LIN {X 0,Y 410.175,Z 395.355,A -85,B 0,C 180,E1 -10523.613,E2 -10523.613} C_VEL
LIN {X 0,Y 410.092,Z 398.974,A -85,B 0,C 180,E1 -10525.084,E2 -10525.084} C_VEL
LIN {X 0,Y 409.955,Z 400.845,A -85,B 0,C 180,E1 -10526.067,E2 -10526.067} C_VEL
LIN {X 0,Y 409.994,Z 402.256,A -85,B 0,C 180,E1 -10527.052,E2 -10527.052} C_VEL
LIN {X 0,Y 409.99,Z 403.255,A -85,B 0,C 180,E1 -10528.035,E2 -10528.035} C_VEL
LIN {X 0,Y 409.957,Z 404.069,A -85,B 0,C 180,E1 -10529.999,E2 -10529.999} C_VEL
LIN {X 0,Y 409.949,Z 403.838,A -85,B 0,C 180,E1 -10530.982,E2 -10530.982} C_VEL
LIN {X 0,Y 409.99,Z 403.212,A -85,B 0,C 180,E1 -10531.964,E2 -10531.964} C_VEL
LIN {X 0,Y 410.009,Z 402.191,A -85,B 0,C 180,E1 -10532.947,E2 -10532.947} C_VEL
LIN {X 0,Y 409.956,Z 400.758,A -85,B 0,C 180,E1 -10533.931,E2 -10533.931} C_VEL
LIN {X 0,Y 410.11,Z 397.769,A -85,B 0,C 180,E1 -10535.408,E2 -10535.408} C_VEL
LIN {X 0,Y 410.201,Z 393.722,A -85,B 0,C 180,E1 -10536.888,E2 -10536.888} C_VEL
LIN {X 0,Y 410.553,Z 387.517,A -85,B 0,C 180,E1 -10538.614,E2 -10538.614} C_VEL
LIN {X 0,Y 410.987,Z 380.75,A -85,B 0,C 180,E1 -10540.094,E2 -10540.094} C_VEL
LIN {X 0,Y 411.568,Z 372.368,A -85,B 0,C 180,E1 -10541.574,E2 -10541.574} C_VEL
LIN {X 0,Y 412.213,Z 363.785,A -85,B 0,C 180,E1 -10542.805,E2 -10542.805} C_VEL
LIN {X 0,Y 412.957,Z 353.054,A -85,B 0,C 180,E1 -10544.051,E2 -10544.051} C_VEL
LIN {X 0,Y 413.774,Z 341.349,A -85,B 0,C 180,E1 -10545.137,E2 -10545.137} C_VEL
LIN {X 0,Y 414.645,Z 329.481,A -85,B 0,C 180,E1 -10545.986,E2 -10545.986} C_VEL
LIN {X 0,Y 414.751,Z 323.251,A -85,B 0,C 180,E1 -10546.359,E2 -10546.359} C_VEL
LIN {X 0,Y 412.959,Z 310.23,A -85,B 0,C 180,E1 -10547.058,E2 -10547.058} C_VEL
LIN {X 0,Y 410.902,Z 297.191,A -85,B 0,C 180,E1 -10547.565,E2 -10547.565} C_VEL
LIN {X 0,Y 410.692,Z 295.43,A -85,B 0,C 180,E1 -10547.629,E2 -10547.629} C_VEL
LIN {X 0,Y 410.997,Z 287.996,A -85,B 0,C 180,E1 -10550.52,E2 -10550.52} C_VEL
LIN {X 0,Y 411.365,Z 280.065,A -85,B 0,C 180,E1 -10553.67,E2 -10553.67} C_VEL
LIN {X 0,Y 411.926,Z 270.899,A -85,B 0,C 180,E1 -10557.429,E2 -10557.429} C_VEL
LIN {X 0,Y 412.494,Z 263.176,A -85,B 0,C 180,E1 -10560.739,E2 -10560.739} C_VEL
LIN {X 0,Y 413.163,Z 255.633,A -85,B 0,C 180,E1 -10564.147,E2 -10564.147} C_VEL
LIN {X 0,Y 413.517,Z 251.98,A -85,B 0,C 180,E1 -10565.897,E2 -10565.897} C_VEL
LIN {X 0,Y 413.199,Z 248.334,A -85,B 0,C 180,E1 -10567.756,E2 -10567.756} C_VEL
LIN {X 0,Y 412.06,Z 241.871,A -85,B 0,C 180,E1 -10571.369,E2 -10571.369} C_VEL
LIN {X 0,Y 411.195,Z 237.269,A -85,B 0,C 180,E1 -10574.262,E2 -10574.262} C_VEL
LIN {X 0,Y 411.193,Z 237.266,A -85,B 0,C 180,E1 -10577.301,E2 -10577.301} C_VEL
LIN {X 0,Y 411.232,Z 237.264,A -85,B 0,C 180,E1 -10580.776,E2 -10580.776} C_VEL
LIN {X 0,Y 411.2,Z 237.268,A -85,B 0,C 180,E1 -10584.47,E2 -10584.47} C_VEL
LIN {X 0,Y 411.207,Z 237.264,A -85,B 0,C 180,E1 -10586.872,E2 -10586.872} C_VEL
LIN {X 0,Y 411.233,Z 237.26,A -85,B 0,C 180,E1 -10590.643,E2 -10590.643} C_VEL
LIN {X 0,Y 411.238,Z 237.261,A -85,B 0,C 180,E1 -10593.618,E2 -10593.618} C_VEL
LIN {X 0,Y 411.202,Z 237.265,A -85,B 0,C 180,E1 -10596.851,E2 -10596.851} C_VEL
LIN {X 0,Y 411.214,Z 237.261,A -85,B 0,C 180,E1 -10600.049,E2 -10600.049} C_VEL
LIN {X 0,Y 411.261,Z 237.258,A -85,B 0,C 180,E1 -10603.13,E2 -10603.13} C_VEL
LIN {X 0,Y 411.303,Z 237.251,A -85,B 0,C 180,E1 -10606.894,E2 -10606.894} C_VEL
LIN {X 0,Y 411.29,Z 237.255,A -85,B 0,C 180,E1 -10610.16,E2 -10610.16} C_VEL
LIN {X 0,Y 411.458,Z 237.233,A -85,B 0,C 180,E1 -10613.131,E2 -10613.131} C_VEL
LIN {X 0,Y 411.309,Z 237.252,A -85,B 0,C 180,E1 -10615.097,E2 -10615.097} C_VEL
LIN {X 0,Y 411.51,Z 237.226,A -85,B 0,C 180,E1 -10618.041,E2 -10618.041} C_VEL
LIN {X 0,Y 411.64,Z 237.211,A -85,B 0,C 180,E1 -10619.998,E2 -10619.998} C_VEL
LIN {X 0,Y 411.461,Z 237.233,A -85,B 0,C 180,E1 -10622.936,E2 -10622.936} C_VEL
LIN {X 0,Y 411.455,Z 237.236,A -85,B 0,C 180,E1 -10626.865,E2 -10626.865} C_VEL
LIN {X 0,Y 411.345,Z 237.249,A -85,B 0,C 180,E1 -10628.844,E2 -10628.844} C_VEL
LIN {X 0,Y 411.165,Z 237.277,A -85,B 0,C 180,E1 -10631.834,E2 -10631.834} C_VEL
LIN {X 0,Y 411.052,Z 237.291,A -85,B 0,C 180,E1 -10632.955,E2 -10632.955} C_VEL
LIN {X 0,Y 410.907,Z 240.592,A -85,B 0,C 180,E1 -10636.707,E2 -10636.707} C_VEL
LIN {X 0,Y 410.742,Z 243.677,A -85,B 0,C 180,E1 -10640.009,E2 -10640.009} C_VEL
LIN {X 0,Y 410.621,Z 246.692,A -85,B 0,C 180,E1 -10643.18,E2 -10643.18} C_VEL
LIN {X 0,Y 410.51,Z 249.844,A -85,B 0,C 180,E1 -10646.429,E2 -10646.429} C_VEL
LIN {X 0,Y 410.442,Z 252.871,A -85,B 0,C 180,E1 -10649.486,E2 -10649.486} C_VEL
LIN {X 0,Y 414.108,Z 266.327,A -85,B 0,C 180,E1 -10650.146,E2 -10650.146} C_VEL
LIN {X 0,Y 415.728,Z 274.254,A -85,B 0,C 180,E1 -10650.613,E2 -10650.613} C_VEL
LIN {X 0,Y 415.069,Z 286.599,A -85,B 0,C 180,E1 -10651.374,E2 -10651.374} C_VEL
LIN {X 0,Y 414.368,Z 298.089,A -85,B 0,C 180,E1 -10652.296,E2 -10652.296} C_VEL
LIN {X 0,Y 413.578,Z 309.114,A -85,B 0,C 180,E1 -10653.422,E2 -10653.422} C_VEL
LIN {X 0,Y 412.865,Z 318.531,A -85,B 0,C 180,E1 -10654.617,E2 -10654.617} C_VEL
LIN {X 0,Y 412.164,Z 327.573,A -85,B 0,C 180,E1 -10656.032,E2 -10656.032} C_VEL
LIN {X 0,Y 411.605,Z 334.198,A -85,B 0,C 180,E1 -10657.308,E2 -10657.308} C_VEL
LIN {X 0,Y 411.016,Z 341.072,A -85,B 0,C 180,E1 -10658.966,E2 -10658.966} C_VEL
LIN {X 0,Y 410.659,Z 346.195,A -85,B 0,C 180,E1 -10660.564,E2 -10660.564} C_VEL
LIN {X 0,Y 410.323,Z 350.805,A -85,B 0,C 180,E1 -10662.567,E2 -10662.567} C_VEL
LIN {X 0,Y 410.109,Z 352.955,A -85,B 0,C 180,E1 -10663.967,E2 -10663.967} C_VEL
LIN {X 0,Y 410.013,Z 354.243,A -85,B 0,C 180,E1 -10665.351,E2 -10665.351} C_VEL
LIN {X 0,Y 409.943,Z 354.715,A -85,B 0,C 180,E1 -10666.706,E2 -10666.706} C_VEL
LIN {X 0,Y 409.959,Z 354.458,A -85,B 0,C 180,E1 -10668.043,E2 -10668.043} C_VEL
LIN {X 0,Y 410.031,Z 353.501,A -85,B 0,C 180,E1 -10669.359,E2 -10669.359} C_VEL
LIN {X 0,Y 410.218,Z 350.71,A -85,B 0,C 180,E1 -10671.294,E2 -10671.294} C_VEL
LIN {X 0,Y 410.512,Z 346.397,A -85,B 0,C 180,E1 -10673.188,E2 -10673.188} C_VEL
LIN {X 0,Y 410.875,Z 341.126,A -85,B 0,C 180,E1 -10674.839,E2 -10674.839} C_VEL
LIN {X 0,Y 411.274,Z 335.33,A -85,B 0,C 180,E1 -10676.265,E2 -10676.265} C_VEL
LIN {X 0,Y 411.887,Z 327.667,A -85,B 0,C 180,E1 -10677.778,E2 -10677.778} C_VEL
LIN {X 0,Y 412.441,Z 320.075,A -85,B 0,C 180,E1 -10679,E2 -10679} C_VEL
LIN {X 0,Y 413.135,Z 310.353,A -85,B 0,C 180,E1 -10680.281,E2 -10680.281} C_VEL
LIN {X 0,Y 413.83,Z 300.496,A -85,B 0,C 180,E1 -10681.331,E2 -10681.331} C_VEL
LIN {X 0,Y 414.563,Z 288.332,A -85,B 0,C 180,E1 -10682.369,E2 -10682.369} C_VEL
LIN {X 0,Y 415.22,Z 276.391,A -85,B 0,C 180,E1 -10683.147,E2 -10683.147} C_VEL
LIN {X 0,Y 415.328,Z 272.584,A -85,B 0,C 180,E1 -10683.358,E2 -10683.358} C_VEL
LIN {X 0,Y 412.637,Z 260.388,A -85,B 0,C 180,E1 -10684.022,E2 -10684.022} C_VEL
LIN {X 0,Y 410.354,Z 251.228,A -85,B 0,C 180,E1 -10684.446,E2 -10684.446} C_VEL
LIN {X 0,Y 410.359,Z 247.606,A -85,B 0,C 180,E1 -10687.866,E2 -10687.866} C_VEL
LIN {X 0,Y 410.438,Z 244.343,A -85,B 0,C 180,E1 -10691.014,E2 -10691.014} C_VEL
LIN {X 0,Y 410.537,Z 241.175,A -85,B 0,C 180,E1 -10694.104,E2 -10694.104} C_VEL
LIN {X 0,Y 410.648,Z 237.964,A -85,B 0,C 180,E1 -10697.285,E2 -10697.285} C_VEL
LIN {X 0,Y 410.713,Z 237.33,A -85,B 0,C 180,E1 -10698.151,E2 -10698.151} C_VEL
LIN {X 0,Y 411.121,Z 237.277,A -85,B 0,C 180,E1 -10701.15,E2 -10701.15} C_VEL
LIN {X 0,Y 411.4,Z 237.241,A -85,B 0,C 180,E1 -10703.133,E2 -10703.133} C_VEL
LIN {X 0,Y 411.299,Z 237.254,A -85,B 0,C 180,E1 -10705.099,E2 -10705.099} C_VEL
LIN {X 0,Y 411.498,Z 237.227,A -85,B 0,C 180,E1 -10708.043,E2 -10708.043} C_VEL
LIN {X 0,Y 411.626,Z 237.21,A -85,B 0,C 180,E1 -10710.006,E2 -10710.006} C_VEL
LIN {X 0,Y 411.452,Z 237.234,A -85,B 0,C 180,E1 -10712.938,E2 -10712.938} C_VEL
LIN {X 0,Y 411.244,Z 237.257,A -85,B 0,C 180,E1 -10714.283,E2 -10714.283} C_VEL
LIN {X 0,Y 410.636,Z 237.337,A -85,B 0,C 180,E1 -10715.101,E2 -10715.101} C_VEL
LIN {X 0,Y 407.876,Z 237.677,A -85,B 0,C 180,E1 -10716.434,E2 -10716.434} C_VEL
LIN {X 0,Y 405.488,Z 237.977,A -85,B 0,C 180,E1 -10717.51,E2 -10717.51} C_VEL
LIN {X 0,Y 404.421,Z 238.107,A -85,B 0,C 180,E1 -10718.34,E2 -10718.34} C_VEL
LIN {X 0,Y 404.314,Z 238.121,A -85,B 0,C 180,E1 -10718.622,E2 -10718.622} C_VEL
LIN {X 0,Y 404.255,Z 238.127,A -85,B 0,C 180,E1 -10722.042,E2 -10722.042} C_VEL
LIN {X 0,Y 404.192,Z 238.139,A -85,B 0,C 180,E1 -10725.119,E2 -10725.119} C_VEL
LIN {X 0,Y 404.199,Z 238.135,A -85,B 0,C 180,E1 -10728.239,E2 -10728.239} C_VEL
LIN {X 0,Y 404.18,Z 238.139,A -85,B 0,C 180,E1 -10731.418,E2 -10731.418} C_VEL
LIN {X 0,Y 404.165,Z 238.143,A -85,B 0,C 180,E1 -10734.667,E2 -10734.667} C_VEL
LIN {X 0,Y 404.182,Z 238.137,A -85,B 0,C 180,E1 -10738.001,E2 -10738.001} C_VEL
LIN {X 0,Y 404.127,Z 238.144,A -85,B 0,C 180,E1 -10741.56,E2 -10741.56} C_VEL
LIN {X 0,Y 404.174,Z 238.141,A -85,B 0,C 180,E1 -10745.018,E2 -10745.018} C_VEL
LIN {X 0,Y 404.153,Z 238.145,A -85,B 0,C 180,E1 -10748.758,E2 -10748.758} C_VEL
LIN {X 0,Y 404.181,Z 238.137,A -85,B 0,C 180,E1 -10751.613,E2 -10751.613} C_VEL
LIN {X 0,Y 404.19,Z 238.14,A -85,B 0,C 180,E1 -10754.532,E2 -10754.532} C_VEL
LIN {X 0,Y 404.202,Z 238.135,A -85,B 0,C 180,E1 -10757.307,E2 -10757.307} C_VEL
LIN {X 0,Y 404.161,Z 238.142,A -85,B 0,C 180,E1 -10759.957,E2 -10759.957} C_VEL
LIN {X 0,Y 404.134,Z 238.143,A -85,B 0,C 180,E1 -10763.126,E2 -10763.126} C_VEL
LIN {X 0,Y 404.139,Z 238.146,A -85,B 0,C 180,E1 -10766.19,E2 -10766.19} C_VEL
LIN {X 0,Y 404.15,Z 238.143,A -85,B 0,C 180,E1 -10769.718,E2 -10769.718} C_VEL
LIN {X 0,Y 404.191,Z 238.135,A -85,B 0,C 180,E1 -10773.125,E2 -10773.125} C_VEL
LIN {X 0,Y 404.174,Z 238.138,A -85,B 0,C 180,E1 -10775.336,E2 -10775.336} C_VEL
LIN {X 0,Y 404.136,Z 238.144,A -85,B 0,C 180,E1 -10778.583,E2 -10778.583} C_VEL
LIN {X 0,Y 404.209,Z 238.136,A -85,B 0,C 180,E1 -10781.764,E2 -10781.764} C_VEL
LIN {X 0,Y 404.205,Z 238.134,A -85,B 0,C 180,E1 -10784.884,E2 -10784.884} C_VEL
LIN {X 0,Y 404.256,Z 238.132,A -85,B 0,C 180,E1 -10787.96,E2 -10787.96} C_VEL
LIN {X 0,Y 404.266,Z 238.126,A -85,B 0,C 180,E1 -10791,E2 -10791} C_VEL
LIN {X 0,Y 404.418,Z 238.112,A -85,B 0,C 180,E1 -10794.017,E2 -10794.017} C_VEL
LIN {X 0,Y 404.482,Z 238.103,A -85,B 0,C 180,E1 -10798.01,E2 -10798.01} C_VEL
LIN {X 0,Y 404.612,Z 238.087,A -85,B 0,C 180,E1 -10800.002,E2 -10800.002} C_VEL
LIN {X 0,Y 404.417,Z 238.108,A -85,B 0,C 180,E1 -10802.99,E2 -10802.99} C_VEL
LIN {X 0,Y 404.373,Z 238.114,A -85,B 0,C 180,E1 -10806.989,E2 -10806.989} C_VEL
LIN {X 0,Y 404.261,Z 238.13,A -85,B 0,C 180,E1 -10810.013,E2 -10810.013} C_VEL
LIN {X 0,Y 404.272,Z 238.128,A -85,B 0,C 180,E1 -10813.213,E2 -10813.213} C_VEL
LIN {X 0,Y 404.221,Z 238.134,A -85,B 0,C 180,E1 -10817.008,E2 -10817.008} C_VEL
LIN {X 0,Y 404.17,Z 238.139,A -85,B 0,C 180,E1 -10820.353,E2 -10820.353} C_VEL
LIN {X 0,Y 404.171,Z 238.143,A -85,B 0,C 180,E1 -10823.576,E2 -10823.576} C_VEL
LIN {X 0,Y 404.187,Z 238.139,A -85,B 0,C 180,E1 -10825.768,E2 -10825.768} C_VEL
LIN {X 0,Y 404.201,Z 238.135,A -85,B 0,C 180,E1 -10828.001,E2 -10828.001} C_VEL
LIN {X 0,Y 404.145,Z 238.145,A -85,B 0,C 180,E1 -10831.559,E2 -10831.559} C_VEL
LIN {X 0,Y 404.19,Z 238.14,A -85,B 0,C 180,E1 -10835.017,E2 -10835.017} C_VEL
LIN {X 0,Y 404.158,Z 238.143,A -85,B 0,C 180,E1 -10838.758,E2 -10838.758} C_VEL
LIN {X 0,Y 404.129,Z 238.145,A -85,B 0,C 180,E1 -10841.6,E2 -10841.6} C_VEL
LIN {X 0,Y 404.152,Z 238.141,A -85,B 0,C 180,E1 -10844.522,E2 -10844.522} C_VEL
LIN {X 0,Y 404.163,Z 238.245,A -85,B 0,C 180,E1 -10846.106,E2 -10846.106} C_VEL
LIN {X 0,Y 405.086,Z 243.048,A -85,B 0,C 180,E1 -10848.755,E2 -10848.755} C_VEL
LIN {X 0,Y 406.008,Z 248.19,A -85,B 0,C 180,E1 -10851.452,E2 -10851.452} C_VEL
LIN {X 0,Y 406.492,Z 252.053,A -85,B 0,C 180,E1 -10853.381,E2 -10853.381} C_VEL
LIN {X 0,Y 406.251,Z 257.069,A -85,B 0,C 180,E1 -10855.73,E2 -10855.73} C_VEL
LIN {X 0,Y 405.685,Z 263.641,A -85,B 0,C 180,E1 -10858.686,E2 -10858.686} C_VEL
LIN {X 0,Y 405.074,Z 271.812,A -85,B 0,C 180,E1 -10862.234,E2 -10862.234} C_VEL
LIN {X 0,Y 404.464,Z 280.525,A -85,B 0,C 180,E1 -10865.899,E2 -10865.899} C_VEL
LIN {X 0,Y 404.05,Z 288.356,A -85,B 0,C 180,E1 -10869.11,E2 -10869.11} C_VEL
LIN {X 0,Y 403.652,Z 295.818,A -85,B 0,C 180,E1 -10872.096,E2 -10872.096} C_VEL
LIN {X 0,Y 405.932,Z 309.766,A -85,B 0,C 180,E1 -10872.631,E2 -10872.631} C_VEL
LIN {X 0,Y 407.729,Z 322.632,A -85,B 0,C 180,E1 -10873.322,E2 -10873.322} C_VEL
LIN {X 0,Y 407.99,Z 325.826,A -85,B 0,C 180,E1 -10873.516,E2 -10873.516} C_VEL
LIN {X 0,Y 407.131,Z 338.126,A -85,B 0,C 180,E1 -10874.352,E2 -10874.352} C_VEL
LIN {X 0,Y 406.279,Z 349.865,A -85,B 0,C 180,E1 -10875.383,E2 -10875.383} C_VEL
LIN {X 0,Y 405.613,Z 359.75,A -85,B 0,C 180,E1 -10876.472,E2 -10876.472} C_VEL
LIN {X 0,Y 404.877,Z 368.986,A -85,B 0,C 180,E1 -10877.722,E2 -10877.722} C_VEL
LIN {X 0,Y 404.108,Z 377.981,A -85,B 0,C 180,E1 -10879.224,E2 -10879.224} C_VEL
LIN {X 0,Y 403.616,Z 385.238,A -85,B 0,C 180,E1 -10880.731,E2 -10880.731} C_VEL
LIN {X 0,Y 403.305,Z 390.139,A -85,B 0,C 180,E1 -10881.986,E2 -10881.986} C_VEL
LIN {X 0,Y 403.068,Z 395.38,A -85,B 0,C 180,E1 -10883.658,E2 -10883.658} C_VEL
LIN {X 0,Y 403.004,Z 398.551,A -85,B 0,C 180,E1 -10884.997,E2 -10884.997} C_VEL
LIN {X 0,Y 402.877,Z 400.424,A -85,B 0,C 180,E1 -10885.998,E2 -10885.998} C_VEL
LIN {X 0,Y 402.897,Z 401.835,A -85,B 0,C 180,E1 -10887,E2 -10887} C_VEL
LIN {X 0,Y 402.922,Z 402.836,A -85,B 0,C 180,E1 -10888,E2 -10888} C_VEL
LIN {X 0,Y 402.881,Z 403.647,A -85,B 0,C 180,E1 -10889.999,E2 -10889.999} C_VEL
LIN {X 0,Y 402.876,Z 403.417,A -85,B 0,C 180,E1 -10890.999,E2 -10890.999} C_VEL
LIN {X 0,Y 402.923,Z 402.79,A -85,B 0,C 180,E1 -10891.999,E2 -10891.999} C_VEL
LIN {X 0,Y 402.91,Z 401.764,A -85,B 0,C 180,E1 -10892.999,E2 -10892.999} C_VEL
LIN {X 0,Y 402.879,Z 400.331,A -85,B 0,C 180,E1 -10894.001,E2 -10894.001} C_VEL
LIN {X 0,Y 403.008,Z 397.336,A -85,B 0,C 180,E1 -10895.503,E2 -10895.503} C_VEL
LIN {X 0,Y 403.12,Z 393.285,A -85,B 0,C 180,E1 -10897.009,E2 -10897.009} C_VEL
LIN {X 0,Y 403.519,Z 387.077,A -85,B 0,C 180,E1 -10898.765,E2 -10898.765} C_VEL
LIN {X 0,Y 403.962,Z 380.309,A -85,B 0,C 180,E1 -10900.272,E2 -10900.272} C_VEL
LIN {X 0,Y 404.577,Z 371.931,A -85,B 0,C 180,E1 -10901.777,E2 -10901.777} C_VEL
LIN {X 0,Y 405.236,Z 363.356,A -85,B 0,C 180,E1 -10903.029,E2 -10903.029} C_VEL
LIN {X 0,Y 405.984,Z 353.509,A -85,B 0,C 180,E1 -10904.203,E2 -10904.203} C_VEL
LIN {X 0,Y 406.781,Z 342.376,A -85,B 0,C 180,E1 -10905.276,E2 -10905.276} C_VEL
LIN {X 0,Y 407.662,Z 331.108,A -85,B 0,C 180,E1 -10906.133,E2 -10906.133} C_VEL
LIN {X 0,Y 407.911,Z 324.517,A -85,B 0,C 180,E1 -10906.549,E2 -10906.549} C_VEL
LIN {X 0,Y 406.181,Z 311.546,A -85,B 0,C 180,E1 -10907.284,E2 -10907.284} C_VEL
LIN {X 0,Y 404.207,Z 298.69,A -85,B 0,C 180,E1 -10907.827,E2 -10907.827} C_VEL
LIN {X 0,Y 403.633,Z 294.95,A -85,B 0,C 180,E1 -10907.969,E2 -10907.969} C_VEL
LIN {X 0,Y 403.947,Z 287.608,A -85,B 0,C 180,E1 -10910.895,E2 -10910.895} C_VEL
LIN {X 0,Y 404.356,Z 279.728,A -85,B 0,C 180,E1 -10914.107,E2 -10914.107} C_VEL
LIN {X 0,Y 404.94,Z 271.136,A -85,B 0,C 180,E1 -10917.73,E2 -10917.73} C_VEL
LIN {X 0,Y 405.485,Z 264.205,A -85,B 0,C 180,E1 -10920.75,E2 -10920.75} C_VEL
LIN {X 0,Y 406.177,Z 256.624,A -85,B 0,C 180,E1 -10924.264,E2 -10924.264} C_VEL
LIN {X 0,Y 406.511,Z 251.844,A -85,B 0,C 180,E1 -10926.616,E2 -10926.616} C_VEL
LIN {X 0,Y 405.905,Z 247.768,A -85,B 0,C 180,E1 -10928.816,E2 -10928.816} C_VEL
LIN {X 0,Y 405,Z 242.759,A -85,B 0,C 180,E1 -10931.738,E2 -10931.738} C_VEL
LIN {X 0,Y 404.148,Z 238.145,A -85,B 0,C 180,E1 -10934.783,E2 -10934.783} C_VEL
LIN {X 0,Y 404.172,Z 238.14,A -85,B 0,C 180,E1 -10937.299,E2 -10937.299} C_VEL
LIN {X 0,Y 404.17,Z 238.141,A -85,B 0,C 180,E1 -10939.954,E2 -10939.954} C_VEL
LIN {X 0,Y 404.141,Z 238.145,A -85,B 0,C 180,E1 -10943.123,E2 -10943.123} C_VEL
LIN {X 0,Y 404.145,Z 238.146,A -85,B 0,C 180,E1 -10946.186,E2 -10946.186} C_VEL
LIN {X 0,Y 404.145,Z 238.145,A -85,B 0,C 180,E1 -10949.713,E2 -10949.713} C_VEL
LIN {X 0,Y 404.195,Z 238.14,A -85,B 0,C 180,E1 -10953.121,E2 -10953.121} C_VEL
LIN {X 0,Y 404.177,Z 238.142,A -85,B 0,C 180,E1 -10955.333,E2 -10955.333} C_VEL
LIN {X 0,Y 404.138,Z 238.146,A -85,B 0,C 180,E1 -10958.579,E2 -10958.579} C_VEL
LIN {X 0,Y 404.209,Z 238.134,A -85,B 0,C 180,E1 -10961.76,E2 -10961.76} C_VEL
LIN {X 0,Y 404.204,Z 238.136,A -85,B 0,C 180,E1 -10964.88,E2 -10964.88} C_VEL
LIN {X 0,Y 404.254,Z 238.132,A -85,B 0,C 180,E1 -10967.957,E2 -10967.957} C_VEL
LIN {X 0,Y 404.43,Z 238.109,A -85,B 0,C 180,E1 -10972.098,E2 -10972.098} C_VEL
LIN {X 0,Y 404.421,Z 238.109,A -85,B 0,C 180,E1 -10974.013,E2 -10974.013} C_VEL
LIN {X 0,Y 404.479,Z 238.101,A -85,B 0,C 180,E1 -10978.007,E2 -10978.007} C_VEL
LIN {X 0,Y 404.609,Z 238.086,A -85,B 0,C 180,E1 -10979.998,E2 -10979.998} C_VEL
LIN {X 0,Y 404.418,Z 238.11,A -85,B 0,C 180,E1 -10982.987,E2 -10982.987} C_VEL
LIN {X 0,Y 404.406,Z 238.113,A -85,B 0,C 180,E1 -10986.986,E2 -10986.986} C_VEL
LIN {X 0,Y 404.235,Z 238.136,A -85,B 0,C 180,E1 -10990.01,E2 -10990.01} C_VEL
LIN {X 0,Y 403.989,Z 238.278,A -85,B 0,C 180,E1 -10993.069,E2 -10993.069} C_VEL
LIN {X 0,Y 403.884,Z 241.052,A -85,B 0,C 180,E1 -10996.164,E2 -10996.164} C_VEL
LIN {X 0,Y 403.74,Z 243.94,A -85,B 0,C 180,E1 -10999.311,E2 -10999.311} C_VEL
LIN {X 0,Y 403.607,Z 247.071,A -85,B 0,C 180,E1 -11002.65,E2 -11002.65} C_VEL
LIN {X 0,Y 403.475,Z 250.084,A -85,B 0,C 180,E1 -11005.813,E2 -11005.813} C_VEL
LIN {X 0,Y 403.398,Z 253.277,A -85,B 0,C 180,E1 -11009.123,E2 -11009.123} C_VEL
LIN {X 0,Y 407.345,Z 267.933,A -85,B 0,C 180,E1 -11009.894,E2 -11009.894} C_VEL
LIN {X 0,Y 408.927,Z 274.744,A -85,B 0,C 180,E1 -11010.32,E2 -11010.32} C_VEL
LIN {X 0,Y 408.285,Z 286.99,A -85,B 0,C 180,E1 -11011.089,E2 -11011.089} C_VEL
LIN {X 0,Y 407.515,Z 299.219,A -85,B 0,C 180,E1 -11012.092,E2 -11012.092} C_VEL
LIN {X 0,Y 406.66,Z 310.427,A -85,B 0,C 180,E1 -11013.276,E2 -11013.276} C_VEL
LIN {X 0,Y 405.847,Z 320.412,A -85,B 0,C 180,E1 -11014.592,E2 -11014.592} C_VEL
LIN {X 0,Y 405.069,Z 329.747,A -85,B 0,C 180,E1 -11016.148,E2 -11016.148} C_VEL
LIN {X 0,Y 404.401,Z 337.233,A -85,B 0,C 180,E1 -11017.711,E2 -11017.711} C_VEL
LIN {X 0,Y 403.851,Z 343.489,A -85,B 0,C 180,E1 -11019.384,E2 -11019.384} C_VEL
LIN {X 0,Y 403.553,Z 347.542,A -85,B 0,C 180,E1 -11020.771,E2 -11020.771} C_VEL
LIN {X 0,Y 403.324,Z 350.608,A -85,B 0,C 180,E1 -11022.131,E2 -11022.131} C_VEL
LIN {X 0,Y 403.199,Z 352.049,A -85,B 0,C 180,E1 -11022.94,E2 -11022.94} C_VEL
LIN {X 0,Y 403.01,Z 353.886,A -85,B 0,C 180,E1 -11024.359,E2 -11024.359} C_VEL
LIN {X 0,Y 402.908,Z 354.9,A -85,B 0,C 180,E1 -11025.756,E2 -11025.756} C_VEL
LIN {X 0,Y 402.859,Z 355.156,A -85,B 0,C 180,E1 -11027.129,E2 -11027.129} C_VEL
LIN {X 0,Y 402.902,Z 354.597,A -85,B 0,C 180,E1 -11028.593,E2 -11028.593} C_VEL
LIN {X 0,Y 402.996,Z 353.094,A -85,B 0,C 180,E1 -11030.111,E2 -11030.111} C_VEL
LIN {X 0,Y 403.194,Z 350.576,A -85,B 0,C 180,E1 -11031.66,E2 -11031.66} C_VEL
LIN {X 0,Y 403.446,Z 346.894,A -85,B 0,C 180,E1 -11033.252,E2 -11033.252} C_VEL
LIN {X 0,Y 403.839,Z 341.573,A -85,B 0,C 180,E1 -11034.95,E2 -11034.95} C_VEL
LIN {X 0,Y 404.317,Z 335.135,A -85,B 0,C 180,E1 -11036.544,E2 -11036.544} C_VEL
LIN {X 0,Y 404.956,Z 327.272,A -85,B 0,C 180,E1 -11038.095,E2 -11038.095} C_VEL
LIN {X 0,Y 405.713,Z 317.918,A -85,B 0,C 180,E1 -11039.558,E2 -11039.558} C_VEL
LIN {X 0,Y 406.436,Z 307.256,A -85,B 0,C 180,E1 -11040.901,E2 -11040.901} C_VEL
LIN {X 0,Y 407.257,Z 296.411,A -85,B 0,C 180,E1 -11041.978,E2 -11041.978} C_VEL
LIN {X 0,Y 407.926,Z 284.699,A -85,B 0,C 180,E1 -11042.905,E2 -11042.905} C_VEL
LIN {X 0,Y 408.486,Z 274.184,A -85,B 0,C 180,E1 -11043.552,E2 -11043.552} C_VEL
LIN {X 0,Y 405.774,Z 261.496,A -85,B 0,C 180,E1 -11044.274,E2 -11044.274} C_VEL
LIN {X 0,Y 403.282,Z 251.628,A -85,B 0,C 180,E1 -11044.725,E2 -11044.725} C_VEL
LIN {X 0,Y 403.276,Z 247.654,A -85,B 0,C 180,E1 -11048.533,E2 -11048.533} C_VEL
LIN {X 0,Y 403.388,Z 244.363,A -85,B 0,C 180,E1 -11051.724,E2 -11051.724} C_VEL
LIN {X 0,Y 403.454,Z 241.195,A -85,B 0,C 180,E1 -11054.854,E2 -11054.854} C_VEL
LIN {X 0,Y 403.639,Z 238.211,A -85,B 0,C 180,E1 -11057.94,E2 -11057.94} C_VEL
LIN {X 0,Y 404.055,Z 238.156,A -85,B 0,C 180,E1 -11060.994,E2 -11060.994} C_VEL
LIN {X 0,Y 404.338,Z 238.12,A -85,B 0,C 180,E1 -11063.012,E2 -11063.012} C_VEL
LIN {X 0,Y 404.27,Z 238.129,A -85,B 0,C 180,E1 -11065.014,E2 -11065.014} C_VEL
LIN {X 0,Y 404.467,Z 238.102,A -85,B 0,C 180,E1 -11068.009,E2 -11068.009} C_VEL
LIN {X 0,Y 404.597,Z 238.086,A -85,B 0,C 180,E1 -11070.001,E2 -11070.001} C_VEL
LIN {X 0,Y 404.409,Z 238.112,A -85,B 0,C 180,E1 -11072.989,E2 -11072.989} C_VEL
LIN {X 0,Y 404.397,Z 238.114,A -85,B 0,C 180,E1 -11076.988,E2 -11076.988} C_VEL
LIN {X 0,Y 404.314,Z 238.121,A -85,B 0,C 180,E1 -11078.622,E2 -11078.622} C_VEL
LIN {X 0,Y 403.583,Z 238.216,A -85,B 0,C 180,E1 -11079.452,E2 -11079.452} C_VEL
LIN {X 0,Y 400.687,Z 238.575,A -85,B 0,C 180,E1 -11080.803,E2 -11080.803} C_VEL
LIN {X 0,Y 398.284,Z 238.871,A -85,B 0,C 180,E1 -11081.893,E2 -11081.893} C_VEL
LIN {X 0,Y 397.274,Z 239,A -85,B 0,C 180,E1 -11082.737,E2 -11082.737} C_VEL
LIN {X 0,Y 397.201,Z 239.008,A -85,B 0,C 180,E1 -11083.022,E2 -11083.022} C_VEL
LIN {X 0,Y 397.151,Z 239.014,A -85,B 0,C 180,E1 -11086.448,E2 -11086.448} C_VEL
LIN {X 0,Y 397.16,Z 239.012,A -85,B 0,C 180,E1 -11089.647,E2 -11089.647} C_VEL
LIN {X 0,Y 397.153,Z 239.017,A -85,B 0,C 180,E1 -11093.053,E2 -11093.053} C_VEL
LIN {X 0,Y 397.123,Z 239.018,A -85,B 0,C 180,E1 -11096.26,E2 -11096.26} C_VEL
LIN {X 0,Y 397.109,Z 239.022,A -85,B 0,C 180,E1 -11098.545,E2 -11098.545} C_VEL
LIN {X 0,Y 397.066,Z 239.024,A -85,B 0,C 180,E1 -11102.073,E2 -11102.073} C_VEL
LIN {X 0,Y 397.109,Z 239.018,A -85,B 0,C 180,E1 -11105.505,E2 -11105.505} C_VEL
LIN {X 0,Y 397.127,Z 239.019,A -85,B 0,C 180,E1 -11108.865,E2 -11108.865} C_VEL
LIN {X 0,Y 397.149,Z 239.016,A -85,B 0,C 180,E1 -11112.257,E2 -11112.257} C_VEL
LIN {X 0,Y 397.142,Z 239.015,A -85,B 0,C 180,E1 -11115.061,E2 -11115.061} C_VEL
LIN {X 0,Y 397.148,Z 239.015,A -85,B 0,C 180,E1 -11118.009,E2 -11118.009} C_VEL
LIN {X 0,Y 397.103,Z 239.019,A -85,B 0,C 180,E1 -11121.728,E2 -11121.728} C_VEL
LIN {X 0,Y 397.12,Z 239.017,A -85,B 0,C 180,E1 -11125.509,E2 -11125.509} C_VEL
LIN {X 0,Y 397.081,Z 239.022,A -85,B 0,C 180,E1 -11129.12,E2 -11129.12} C_VEL
LIN {X 0,Y 397.191,Z 239.01,A -85,B 0,C 180,E1 -11132.612,E2 -11132.612} C_VEL
LIN {X 0,Y 397.13,Z 239.019,A -85,B 0,C 180,E1 -11135.984,E2 -11135.984} C_VEL
LIN {X 0,Y 397.136,Z 239.016,A -85,B 0,C 180,E1 -11139.707,E2 -11139.707} C_VEL
LIN {X 0,Y 397.181,Z 239.009,A -85,B 0,C 180,E1 -11142.847,E2 -11142.847} C_VEL
LIN {X 0,Y 397.228,Z 239.004,A -85,B 0,C 180,E1 -11146.705,E2 -11146.705} C_VEL
LIN {X 0,Y 397.217,Z 239.008,A -85,B 0,C 180,E1 -11149.811,E2 -11149.811} C_VEL
LIN {X 0,Y 397.336,Z 238.99,A -85,B 0,C 180,E1 -11152.89,E2 -11152.89} C_VEL
LIN {X 0,Y 397.254,Z 239,A -85,B 0,C 180,E1 -11154.927,E2 -11154.927} C_VEL
LIN {X 0,Y 397.451,Z 238.979,A -85,B 0,C 180,E1 -11157.975,E2 -11157.975} C_VEL
LIN {X 0,Y 397.581,Z 238.962,A -85,B 0,C 180,E1 -11160.002,E2 -11160.002} C_VEL
LIN {X 0,Y 397.376,Z 238.985,A -85,B 0,C 180,E1 -11163.043,E2 -11163.043} C_VEL
LIN {X 0,Y 397.348,Z 238.99,A -85,B 0,C 180,E1 -11166.094,E2 -11166.094} C_VEL
LIN {X 0,Y 397.24,Z 239.004,A -85,B 0,C 180,E1 -11169.164,E2 -11169.164} C_VEL
LIN {X 0,Y 397.224,Z 239.004,A -85,B 0,C 180,E1 -11172.26,E2 -11172.26} C_VEL
LIN {X 0,Y 397.184,Z 239.012,A -85,B 0,C 180,E1 -11175.393,E2 -11175.393} C_VEL
LIN {X 0,Y 397.168,Z 239.01,A -85,B 0,C 180,E1 -11178.575,E2 -11178.575} C_VEL
LIN {X 0,Y 397.103,Z 239.021,A -85,B 0,C 180,E1 -11181.82,E2 -11181.82} C_VEL
LIN {X 0,Y 397.161,Z 239.015,A -85,B 0,C 180,E1 -11185.133,E2 -11185.133} C_VEL
LIN {X 0,Y 397.168,Z 239.012,A -85,B 0,C 180,E1 -11187.777,E2 -11187.777} C_VEL
LIN {X 0,Y 397.085,Z 239.023,A -85,B 0,C 180,E1 -11190.883,E2 -11190.883} C_VEL
LIN {X 0,Y 397.131,Z 239.016,A -85,B 0,C 180,E1 -11194.494,E2 -11194.494} C_VEL
LIN {X 0,Y 397.107,Z 239.022,A -85,B 0,C 180,E1 -11198.276,E2 -11198.276} C_VEL
LIN {X 0,Y 397.095,Z 239.024,A -85,B 0,C 180,E1 -11200.909,E2 -11200.909} C_VEL
LIN {X 0,Y 397.108,Z 239.017,A -85,B 0,C 180,E1 -11203.649,E2 -11203.649} C_VEL
LIN {X 0,Y 397.116,Z 239.098,A -85,B 0,C 180,E1 -11205.734,E2 -11205.734} C_VEL
LIN {X 0,Y 398.326,Z 245.561,A -85,B 0,C 180,E1 -11209.35,E2 -11209.35} C_VEL
LIN {X 0,Y 399.309,Z 251.32,A -85,B 0,C 180,E1 -11212.376,E2 -11212.376} C_VEL
LIN {X 0,Y 399.475,Z 255.661,A -85,B 0,C 180,E1 -11214.509,E2 -11214.509} C_VEL
LIN {X 0,Y 398.801,Z 263.353,A -85,B 0,C 180,E1 -11218.083,E2 -11218.083} C_VEL
LIN {X 0,Y 398.08,Z 272.12,A -85,B 0,C 180,E1 -11221.976,E2 -11221.976} C_VEL
LIN {X 0,Y 397.46,Z 280.202,A -85,B 0,C 180,E1 -11225.447,E2 -11225.447} C_VEL
LIN {X 0,Y 396.998,Z 287.992,A -85,B 0,C 180,E1 -11228.721,E2 -11228.721} C_VEL
LIN {X 0,Y 396.625,Z 295.512,A -85,B 0,C 180,E1 -11231.785,E2 -11231.785} C_VEL
LIN {X 0,Y 398.843,Z 309.348,A -85,B 0,C 180,E1 -11232.32,E2 -11232.32} C_VEL
LIN {X 0,Y 400.72,Z 322.711,A -85,B 0,C 180,E1 -11233.059,E2 -11233.059} C_VEL
LIN {X 0,Y 401.032,Z 327.493,A -85,B 0,C 180,E1 -11233.365,E2 -11233.365} C_VEL
LIN {X 0,Y 400.155,Z 339.194,A -85,B 0,C 180,E1 -11234.203,E2 -11234.203} C_VEL
LIN {X 0,Y 399.274,Z 350.754,A -85,B 0,C 180,E1 -11235.265,E2 -11235.265} C_VEL
LIN {X 0,Y 398.479,Z 361.305,A -85,B 0,C 180,E1 -11236.493,E2 -11236.493} C_VEL
LIN {X 0,Y 397.752,Z 370.16,A -85,B 0,C 180,E1 -11237.758,E2 -11237.758} C_VEL
LIN {X 0,Y 396.989,Z 378.875,A -85,B 0,C 180,E1 -11239.287,E2 -11239.287} C_VEL
LIN {X 0,Y 396.502,Z 385.839,A -85,B 0,C 180,E1 -11240.82,E2 -11240.82} C_VEL
LIN {X 0,Y 396.142,Z 391.422,A -85,B 0,C 180,E1 -11242.353,E2 -11242.353} C_VEL
LIN {X 0,Y 395.955,Z 395.806,A -85,B 0,C 180,E1 -11243.886,E2 -11243.886} C_VEL
LIN {X 0,Y 395.917,Z 398.125,A -85,B 0,C 180,E1 -11244.907,E2 -11244.907} C_VEL
LIN {X 0,Y 395.802,Z 400.001,A -85,B 0,C 180,E1 -11245.927,E2 -11245.927} C_VEL
LIN {X 0,Y 395.8,Z 401.412,A -85,B 0,C 180,E1 -11246.946,E2 -11246.946} C_VEL
LIN {X 0,Y 395.855,Z 402.415,A -85,B 0,C 180,E1 -11247.965,E2 -11247.965} C_VEL
LIN {X 0,Y 395.806,Z 403.226,A -85,B 0,C 180,E1 -11249.999,E2 -11249.999} C_VEL
LIN {X 0,Y 395.805,Z 402.995,A -85,B 0,C 180,E1 -11251.017,E2 -11251.017} C_VEL
LIN {X 0,Y 395.856,Z 402.367,A -85,B 0,C 180,E1 -11252.034,E2 -11252.034} C_VEL
LIN {X 0,Y 395.813,Z 401.339,A -85,B 0,C 180,E1 -11253.053,E2 -11253.053} C_VEL
LIN {X 0,Y 395.804,Z 399.906,A -85,B 0,C 180,E1 -11254.072,E2 -11254.072} C_VEL
LIN {X 0,Y 395.909,Z 396.908,A -85,B 0,C 180,E1 -11255.602,E2 -11255.602} C_VEL
LIN {X 0,Y 396.065,Z 392.859,A -85,B 0,C 180,E1 -11257.135,E2 -11257.135} C_VEL
LIN {X 0,Y 396.46,Z 386.653,A -85,B 0,C 180,E1 -11258.923,E2 -11258.923} C_VEL
LIN {X 0,Y 396.912,Z 379.883,A -85,B 0,C 180,E1 -11260.456,E2 -11260.456} C_VEL
LIN {X 0,Y 397.572,Z 371.506,A -85,B 0,C 180,E1 -11261.987,E2 -11261.987} C_VEL
LIN {X 0,Y 398.286,Z 362.945,A -85,B 0,C 180,E1 -11263.261,E2 -11263.261} C_VEL
LIN {X 0,Y 399.099,Z 352.639,A -85,B 0,C 180,E1 -11264.506,E2 -11264.506} C_VEL
LIN {X 0,Y 399.93,Z 342.013,A -85,B 0,C 180,E1 -11265.544,E2 -11265.544} C_VEL
LIN {X 0,Y 400.82,Z 330.862,A -85,B 0,C 180,E1 -11266.41,E2 -11266.41} C_VEL
LIN {X 0,Y 401.048,Z 325.611,A -85,B 0,C 180,E1 -11266.754,E2 -11266.754} C_VEL
LIN {X 0,Y 399.398,Z 312.798,A -85,B 0,C 180,E1 -11267.523,E2 -11267.523} C_VEL
LIN {X 0,Y 397.441,Z 299.565,A -85,B 0,C 180,E1 -11268.116,E2 -11268.116} C_VEL
LIN {X 0,Y 396.612,Z 294.561,A -85,B 0,C 180,E1 -11268.298,E2 -11268.298} C_VEL
LIN {X 0,Y 396.918,Z 287.232,A -85,B 0,C 180,E1 -11271.283,E2 -11271.283} C_VEL
LIN {X 0,Y 397.37,Z 279.389,A -85,B 0,C 180,E1 -11274.558,E2 -11274.558} C_VEL
LIN {X 0,Y 397.956,Z 271.456,A -85,B 0,C 180,E1 -11277.99,E2 -11277.99} C_VEL
LIN {X 0,Y 398.535,Z 264.031,A -85,B 0,C 180,E1 -11281.346,E2 -11281.346} C_VEL
LIN {X 0,Y 399.193,Z 257.814,A -85,B 0,C 180,E1 -11284.289,E2 -11284.289} C_VEL
LIN {X 0,Y 399.528,Z 254.366,A -85,B 0,C 180,E1 -11285.983,E2 -11285.983} C_VEL
LIN {X 0,Y 399.199,Z 250.555,A -85,B 0,C 180,E1 -11288.037,E2 -11288.037} C_VEL
LIN {X 0,Y 398.164,Z 244.754,A -85,B 0,C 180,E1 -11291.427,E2 -11291.427} C_VEL
LIN {X 0,Y 397.144,Z 239.394,A -85,B 0,C 180,E1 -11294.938,E2 -11294.938} C_VEL
LIN {X 0,Y 397.098,Z 239.024,A -85,B 0,C 180,E1 -11295.386,E2 -11295.386} C_VEL
LIN {X 0,Y 397.111,Z 239.022,A -85,B 0,C 180,E1 -11298.013,E2 -11298.013} C_VEL
LIN {X 0,Y 397.139,Z 239.019,A -85,B 0,C 180,E1 -11301.136,E2 -11301.136} C_VEL
LIN {X 0,Y 397.12,Z 239.022,A -85,B 0,C 180,E1 -11304.495,E2 -11304.495} C_VEL
LIN {X 0,Y 397.079,Z 239.027,A -85,B 0,C 180,E1 -11307.927,E2 -11307.927} C_VEL
LIN {X 0,Y 397.122,Z 239.019,A -85,B 0,C 180,E1 -11311.455,E2 -11311.455} C_VEL
LIN {X 0,Y 397.152,Z 239.016,A -85,B 0,C 180,E1 -11314.486,E2 -11314.486} C_VEL
LIN {X 0,Y 397.108,Z 239.02,A -85,B 0,C 180,E1 -11317.084,E2 -11317.084} C_VEL
LIN {X 0,Y 397.147,Z 239.014,A -85,B 0,C 180,E1 -11320.351,E2 -11320.351} C_VEL
LIN {X 0,Y 397.165,Z 239.015,A -85,B 0,C 180,E1 -11323.552,E2 -11323.552} C_VEL
LIN {X 0,Y 397.226,Z 239.004,A -85,B 0,C 180,E1 -11326.701,E2 -11326.701} C_VEL
LIN {X 0,Y 397.215,Z 239.007,A -85,B 0,C 180,E1 -11329.807,E2 -11329.807} C_VEL
LIN {X 0,Y 397.361,Z 238.99,A -85,B 0,C 180,E1 -11332.887,E2 -11332.887} C_VEL
LIN {X 0,Y 397.253,Z 239.004,A -85,B 0,C 180,E1 -11334.924,E2 -11334.924} C_VEL
LIN {X 0,Y 397.448,Z 238.977,A -85,B 0,C 180,E1 -11337.972,E2 -11337.972} C_VEL
LIN {X 0,Y 397.578,Z 238.962,A -85,B 0,C 180,E1 -11339.998,E2 -11339.998} C_VEL
LIN {X 0,Y 397.376,Z 238.988,A -85,B 0,C 180,E1 -11343.04,E2 -11343.04} C_VEL
LIN {X 0,Y 397.358,Z 238.991,A -85,B 0,C 180,E1 -11347.11,E2 -11347.11} C_VEL
LIN {X 0,Y 397.19,Z 239.014,A -85,B 0,C 180,E1 -11350.19,E2 -11350.19} C_VEL
LIN {X 0,Y 397.026,Z 239.039,A -85,B 0,C 180,E1 -11352.262,E2 -11352.262} C_VEL
LIN {X 0,Y 396.94,Z 239.513,A -85,B 0,C 180,E1 -11353.305,E2 -11353.305} C_VEL
LIN {X 0,Y 396.821,Z 242.782,A -85,B 0,C 180,E1 -11356.988,E2 -11356.988} C_VEL
LIN {X 0,Y 396.655,Z 245.618,A -85,B 0,C 180,E1 -11360.108,E2 -11360.108} C_VEL
LIN {X 0,Y 396.562,Z 248.238,A -85,B 0,C 180,E1 -11362.945,E2 -11362.945} C_VEL
LIN {X 0,Y 396.417,Z 251.417,A -85,B 0,C 180,E1 -11366.307,E2 -11366.307} C_VEL
LIN {X 0,Y 396.35,Z 253.778,A -85,B 0,C 180,E1 -11368.783,E2 -11368.783} C_VEL
LIN {X 0,Y 400.351,Z 268.179,A -85,B 0,C 180,E1 -11369.552,E2 -11369.552} C_VEL
LIN {X 0,Y 402.172,Z 276.569,A -85,B 0,C 180,E1 -11370.094,E2 -11370.094} C_VEL
LIN {X 0,Y 401.433,Z 289.192,A -85,B 0,C 180,E1 -11370.925,E2 -11370.925} C_VEL
LIN {X 0,Y 400.64,Z 300.336,A -85,B 0,C 180,E1 -11371.881,E2 -11371.881} C_VEL
LIN {X 0,Y 399.795,Z 310.86,A -85,B 0,C 180,E1 -11373.019,E2 -11373.019} C_VEL
LIN {X 0,Y 398.984,Z 320.506,A -85,B 0,C 180,E1 -11374.307,E2 -11374.307} C_VEL
LIN {X 0,Y 398.248,Z 329.094,A -85,B 0,C 180,E1 -11375.732,E2 -11375.732} C_VEL
LIN {X 0,Y 397.522,Z 336.646,A -85,B 0,C 180,E1 -11377.291,E2 -11377.291} C_VEL
LIN {X 0,Y 396.953,Z 342.594,A -85,B 0,C 180,E1 -11378.831,E2 -11378.831} C_VEL
LIN {X 0,Y 396.564,Z 347.224,A -85,B 0,C 180,E1 -11380.355,E2 -11380.355} C_VEL
LIN {X 0,Y 396.205,Z 351.686,A -85,B 0,C 180,E1 -11382.378,E2 -11382.378} C_VEL
LIN {X 0,Y 395.982,Z 353.802,A -85,B 0,C 180,E1 -11383.8,E2 -11383.8} C_VEL
LIN {X 0,Y 395.858,Z 355.103,A -85,B 0,C 180,E1 -11385.244,E2 -11385.244} C_VEL
LIN {X 0,Y 395.765,Z 355.591,A -85,B 0,C 180,E1 -11386.722,E2 -11386.722} C_VEL
LIN {X 0,Y 395.795,Z 355.231,A -85,B 0,C 180,E1 -11388.223,E2 -11388.223} C_VEL
LIN {X 0,Y 395.926,Z 353.349,A -85,B 0,C 180,E1 -11390.282,E2 -11390.282} C_VEL
LIN {X 0,Y 396.211,Z 349.87,A -85,B 0,C 180,E1 -11392.269,E2 -11392.269} C_VEL
LIN {X 0,Y 396.604,Z 344.823,A -85,B 0,C 180,E1 -11394.214,E2 -11394.214} C_VEL
LIN {X 0,Y 397.045,Z 338.819,A -85,B 0,C 180,E1 -11395.919,E2 -11395.919} C_VEL
LIN {X 0,Y 397.606,Z 332.339,A -85,B 0,C 180,E1 -11397.378,E2 -11397.378} C_VEL
LIN {X 0,Y 398.27,Z 323.839,A -85,B 0,C 180,E1 -11398.926,E2 -11398.926} C_VEL
LIN {X 0,Y 398.991,Z 315.085,A -85,B 0,C 180,E1 -11400.208,E2 -11400.208} C_VEL
LIN {X 0,Y 399.812,Z 304.129,A -85,B 0,C 180,E1 -11401.506,E2 -11401.506} C_VEL
LIN {X 0,Y 400.642,Z 292.641,A -85,B 0,C 180,E1 -11402.583,E2 -11402.583} C_VEL
LIN {X 0,Y 401.39,Z 280.011,A -85,B 0,C 180,E1 -11403.499,E2 -11403.499} C_VEL
LIN {X 0,Y 401.55,Z 274.842,A -85,B 0,C 180,E1 -11403.808,E2 -11403.808} C_VEL
LIN {X 0,Y 398.889,Z 262.513,A -85,B 0,C 180,E1 -11404.532,E2 -11404.532} C_VEL
LIN {X 0,Y 396.215,Z 252.027,A -85,B 0,C 180,E1 -11405.016,E2 -11405.016} C_VEL
LIN {X 0,Y 396.2,Z 248.801,A -85,B 0,C 180,E1 -11408.13,E2 -11408.13} C_VEL
LIN {X 0,Y 396.311,Z 245.465,A -85,B 0,C 180,E1 -11411.386,E2 -11411.386} C_VEL
LIN {X 0,Y 396.391,Z 242.265,A -85,B 0,C 180,E1 -11414.577,E2 -11414.577} C_VEL
LIN {X 0,Y 396.559,Z 239.151,A -85,B 0,C 180,E1 -11417.722,E2 -11417.722} C_VEL
LIN {X 0,Y 396.984,Z 239.035,A -85,B 0,C 180,E1 -11420.833,E2 -11420.833} C_VEL
LIN {X 0,Y 397.278,Z 238.999,A -85,B 0,C 180,E1 -11422.887,E2 -11422.887} C_VEL
LIN {X 0,Y 397.241,Z 239.004,A -85,B 0,C 180,E1 -11424.926,E2 -11424.926} C_VEL
LIN {X 0,Y 397.436,Z 238.978,A -85,B 0,C 180,E1 -11427.974,E2 -11427.974} C_VEL
LIN {X 0,Y 397.566,Z 238.961,A -85,B 0,C 180,E1 -11430.001,E2 -11430.001} C_VEL
LIN {X 0,Y 397.368,Z 238.989,A -85,B 0,C 180,E1 -11433.042,E2 -11433.042} C_VEL
LIN {X 0,Y 397.349,Z 238.992,A -85,B 0,C 180,E1 -11437.113,E2 -11437.113} C_VEL
LIN {X 0,Y 397.214,Z 239.005,A -85,B 0,C 180,E1 -11440.192,E2 -11440.192} C_VEL
LIN {X 0,Y 397.201,Z 239.008,A -85,B 0,C 180,E1 -11443.022,E2 -11443.022} C_VEL
LIN {X 0,Y 396.558,Z 239.093,A -85,B 0,C 180,E1 -11443.868,E2 -11443.868} C_VEL
LIN {X 0,Y 393.71,Z 239.451,A -85,B 0,C 180,E1 -11445.243,E2 -11445.243} C_VEL
LIN {X 0,Y 391.275,Z 239.752,A -85,B 0,C 180,E1 -11446.354,E2 -11446.354} C_VEL
LIN {X 0,Y 390.216,Z 239.88,A -85,B 0,C 180,E1 -11447.213,E2 -11447.213} C_VEL
LIN {X 0,Y 390.123,Z 239.889,A -85,B 0,C 180,E1 -11447.504,E2 -11447.504} C_VEL
LIN {X 0,Y 390.091,Z 239.895,A -85,B 0,C 180,E1 -11451.121,E2 -11451.121} C_VEL
LIN {X 0,Y 390.071,Z 239.896,A -85,B 0,C 180,E1 -11454.482,E2 -11454.482} C_VEL
LIN {X 0,Y 390.104,Z 239.89,A -85,B 0,C 180,E1 -11457.931,E2 -11457.931} C_VEL
LIN {X 0,Y 390.011,Z 239.902,A -85,B 0,C 180,E1 -11461.506,E2 -11461.506} C_VEL
LIN {X 0,Y 390.074,Z 239.895,A -85,B 0,C 180,E1 -11465.209,E2 -11465.209} C_VEL
LIN {X 0,Y 390.085,Z 239.895,A -85,B 0,C 180,E1 -11469.093,E2 -11469.093} C_VEL
LIN {X 0,Y 390.111,Z 239.893,A -85,B 0,C 180,E1 -11472.389,E2 -11472.389} C_VEL
LIN {X 0,Y 390.11,Z 239.889,A -85,B 0,C 180,E1 -11475.367,E2 -11475.367} C_VEL
LIN {X 0,Y 390.097,Z 239.894,A -85,B 0,C 180,E1 -11478.198,E2 -11478.198} C_VEL
LIN {X 0,Y 390.088,Z 239.894,A -85,B 0,C 180,E1 -11480.91,E2 -11480.91} C_VEL
LIN {X 0,Y 390.079,Z 239.896,A -85,B 0,C 180,E1 -11484.795,E2 -11484.795} C_VEL
LIN {X 0,Y 390.042,Z 239.902,A -85,B 0,C 180,E1 -11488.5,E2 -11488.5} C_VEL
LIN {X 0,Y 390.113,Z 239.893,A -85,B 0,C 180,E1 -11492.072,E2 -11492.072} C_VEL
LIN {X 0,Y 390.077,Z 239.895,A -85,B 0,C 180,E1 -11495.521,E2 -11495.521} C_VEL
LIN {X 0,Y 390.053,Z 239.896,A -85,B 0,C 180,E1 -11498.88,E2 -11498.88} C_VEL
LIN {X 0,Y 390.127,Z 239.892,A -85,B 0,C 180,E1 -11502.169,E2 -11502.169} C_VEL
LIN {X 0,Y 390.143,Z 239.886,A -85,B 0,C 180,E1 -11505.395,E2 -11505.395} C_VEL
LIN {X 0,Y 390.147,Z 239.886,A -85,B 0,C 180,E1 -11508.573,E2 -11508.573} C_VEL
LIN {X 0,Y 390.271,Z 239.873,A -85,B 0,C 180,E1 -11512.073,E2 -11512.073} C_VEL
LIN {X 0,Y 390.226,Z 239.875,A -85,B 0,C 180,E1 -11514.835,E2 -11514.835} C_VEL
LIN {X 0,Y 390.42,Z 239.855,A -85,B 0,C 180,E1 -11517.939,E2 -11517.939} C_VEL
LIN {X 0,Y 390.551,Z 239.838,A -85,B 0,C 180,E1 -11520.002,E2 -11520.002} C_VEL
LIN {X 0,Y 390.311,Z 239.866,A -85,B 0,C 180,E1 -11523.098,E2 -11523.098} C_VEL
LIN {X 0,Y 390.302,Z 239.867,A -85,B 0,C 180,E1 -11526.204,E2 -11526.204} C_VEL
LIN {X 0,Y 390.197,Z 239.882,A -85,B 0,C 180,E1 -11529.331,E2 -11529.331} C_VEL
LIN {X 0,Y 390.175,Z 239.881,A -85,B 0,C 180,E1 -11532.485,E2 -11532.485} C_VEL
LIN {X 0,Y 390.145,Z 239.889,A -85,B 0,C 180,E1 -11535.678,E2 -11535.678} C_VEL
LIN {X 0,Y 390.111,Z 239.89,A -85,B 0,C 180,E1 -11538.923,E2 -11538.923} C_VEL
LIN {X 0,Y 390.045,Z 239.898,A -85,B 0,C 180,E1 -11542.235,E2 -11542.235} C_VEL
LIN {X 0,Y 390.123,Z 239.89,A -85,B 0,C 180,E1 -11545.744,E2 -11545.744} C_VEL
LIN {X 0,Y 390.065,Z 239.899,A -85,B 0,C 180,E1 -11549.111,E2 -11549.111} C_VEL
LIN {X 0,Y 390.049,Z 239.899,A -85,B 0,C 180,E1 -11552.722,E2 -11552.722} C_VEL
LIN {X 0,Y 390.062,Z 239.896,A -85,B 0,C 180,E1 -11555.826,E2 -11555.826} C_VEL
LIN {X 0,Y 390.074,Z 239.898,A -85,B 0,C 180,E1 -11559.219,E2 -11559.219} C_VEL
LIN {X 0,Y 390.049,Z 239.897,A -85,B 0,C 180,E1 -11562.375,E2 -11562.375} C_VEL
LIN {X 0,Y 390.076,Z 239.937,A -85,B 0,C 180,E1 -11565.358,E2 -11565.358} C_VEL
LIN {X 0,Y 391.25,Z 246.271,A -85,B 0,C 180,E1 -11568.978,E2 -11568.978} C_VEL
LIN {X 0,Y 392.253,Z 251.925,A -85,B 0,C 180,E1 -11572.033,E2 -11572.033} C_VEL
LIN {X 0,Y 392.51,Z 255.367,A -85,B 0,C 180,E1 -11573.78,E2 -11573.78} C_VEL
LIN {X 0,Y 392.118,Z 260.499,A -85,B 0,C 180,E1 -11576.246,E2 -11576.246} C_VEL
LIN {X 0,Y 391.651,Z 265.629,A -85,B 0,C 180,E1 -11578.641,E2 -11578.641} C_VEL
LIN {X 0,Y 390.978,Z 273.374,A -85,B 0,C 180,E1 -11582.136,E2 -11582.136} C_VEL
LIN {X 0,Y 390.374,Z 281.129,A -85,B 0,C 180,E1 -11585.538,E2 -11585.538} C_VEL
LIN {X 0,Y 389.92,Z 288.91,A -85,B 0,C 180,E1 -11588.87,E2 -11588.87} C_VEL
LIN {X 0,Y 389.567,Z 295.291,A -85,B 0,C 180,E1 -11591.46,E2 -11591.46} C_VEL
LIN {X 0,Y 391.86,Z 309.041,A -85,B 0,C 180,E1 -11592.012,E2 -11592.012} C_VEL
LIN {X 0,Y 393.598,Z 321.83,A -85,B 0,C 180,E1 -11592.727,E2 -11592.727} C_VEL
LIN {X 0,Y 394.175,Z 327.25,A -85,B 0,C 180,E1 -11593.089,E2 -11593.089} C_VEL
LIN {X 0,Y 393.306,Z 338.657,A -85,B 0,C 180,E1 -11593.92,E2 -11593.92} C_VEL
LIN {X 0,Y 392.414,Z 349.756,A -85,B 0,C 180,E1 -11594.948,E2 -11594.948} C_VEL
LIN {X 0,Y 391.69,Z 359.32,A -85,B 0,C 180,E1 -11596.052,E2 -11596.052} C_VEL
LIN {X 0,Y 390.965,Z 368.055,A -85,B 0,C 180,E1 -11597.278,E2 -11597.278} C_VEL
LIN {X 0,Y 390.083,Z 377.069,A -85,B 0,C 180,E1 -11598.832,E2 -11598.832} C_VEL
LIN {X 0,Y 389.548,Z 384.345,A -85,B 0,C 180,E1 -11600.393,E2 -11600.393} C_VEL
LIN {X 0,Y 389.184,Z 389.258,A -85,B 0,C 180,E1 -11601.693,E2 -11601.693} C_VEL
LIN {X 0,Y 388.92,Z 394.037,A -85,B 0,C 180,E1 -11603.255,E2 -11603.255} C_VEL
LIN {X 0,Y 388.831,Z 397.691,A -85,B 0,C 180,E1 -11604.814,E2 -11604.814} C_VEL
LIN {X 0,Y 388.729,Z 399.571,A -85,B 0,C 180,E1 -11605.852,E2 -11605.852} C_VEL
LIN {X 0,Y 388.706,Z 400.985,A -85,B 0,C 180,E1 -11606.89,E2 -11606.89} C_VEL
LIN {X 0,Y 388.788,Z 401.991,A -85,B 0,C 180,E1 -11607.928,E2 -11607.928} C_VEL
LIN {X 0,Y 388.735,Z 402.805,A -85,B 0,C 180,E1 -11609.999,E2 -11609.999} C_VEL
LIN {X 0,Y 388.736,Z 402.576,A -85,B 0,C 180,E1 -11611.035,E2 -11611.035} C_VEL
LIN {X 0,Y 388.79,Z 401.947,A -85,B 0,C 180,E1 -11612.071,E2 -11612.071} C_VEL
LIN {X 0,Y 388.731,Z 399.485,A -85,B 0,C 180,E1 -11614.147,E2 -11614.147} C_VEL
LIN {X 0,Y 388.833,Z 396.035,A -85,B 0,C 180,E1 -11615.898,E2 -11615.898} C_VEL
LIN {X 0,Y 389.081,Z 390.819,A -85,B 0,C 180,E1 -11617.785,E2 -11617.785} C_VEL
LIN {X 0,Y 389.452,Z 385.209,A -85,B 0,C 180,E1 -11619.346,E2 -11619.346} C_VEL
LIN {X 0,Y 389.959,Z 378.221,A -85,B 0,C 180,E1 -11620.908,E2 -11620.908} C_VEL
LIN {X 0,Y 390.784,Z 369.512,A -85,B 0,C 180,E1 -11622.463,E2 -11622.463} C_VEL
LIN {X 0,Y 391.662,Z 359.372,A -85,B 0,C 180,E1 -11623.919,E2 -11623.919} C_VEL
LIN {X 0,Y 392.484,Z 348.413,A -85,B 0,C 180,E1 -11625.181,E2 -11625.181} C_VEL
LIN {X 0,Y 393.462,Z 337.15,A -85,B 0,C 180,E1 -11626.205,E2 -11626.205} C_VEL
LIN {X 0,Y 394.181,Z 327.345,A -85,B 0,C 180,E1 -11626.92,E2 -11626.92} C_VEL
LIN {X 0,Y 392.785,Z 315.12,A -85,B 0,C 180,E1 -11627.708,E2 -11627.708} C_VEL
LIN {X 0,Y 390.954,Z 302.158,A -85,B 0,C 180,E1 -11628.35,E2 -11628.35} C_VEL
LIN {X 0,Y 389.557,Z 294.047,A -85,B 0,C 180,E1 -11628.676,E2 -11628.676} C_VEL
LIN {X 0,Y 389.886,Z 286.867,A -85,B 0,C 180,E1 -11631.686,E2 -11631.686} C_VEL
LIN {X 0,Y 390.382,Z 279.076,A -85,B 0,C 180,E1 -11635.028,E2 -11635.028} C_VEL
LIN {X 0,Y 390.95,Z 271.798,A -85,B 0,C 180,E1 -11638.252,E2 -11638.252} C_VEL
LIN {X 0,Y 391.516,Z 265.038,A -85,B 0,C 180,E1 -11641.37,E2 -11641.37} C_VEL
LIN {X 0,Y 392.341,Z 257.61,A -85,B 0,C 180,E1 -11644.974,E2 -11644.974} C_VEL
LIN {X 0,Y 392.509,Z 254.04,A -85,B 0,C 180,E1 -11646.857,E2 -11646.857} C_VEL
LIN {X 0,Y 391.773,Z 249.372,A -85,B 0,C 180,E1 -11649.521,E2 -11649.521} C_VEL
LIN {X 0,Y 390.898,Z 244.544,A -85,B 0,C 180,E1 -11652.51,E2 -11652.51} C_VEL
LIN {X 0,Y 390.08,Z 239.896,A -85,B 0,C 180,E1 -11655.781,E2 -11655.781} C_VEL
LIN {X 0,Y 390.078,Z 239.898,A -85,B 0,C 180,E1 -11659.174,E2 -11659.174} C_VEL
LIN {X 0,Y 390.048,Z 239.903,A -85,B 0,C 180,E1 -11662.447,E2 -11662.447} C_VEL
LIN {X 0,Y 390.068,Z 239.9,A -85,B 0,C 180,E1 -11666.044,E2 -11666.044} C_VEL
LIN {X 0,Y 390.047,Z 239.902,A -85,B 0,C 180,E1 -11669.867,E2 -11669.867} C_VEL
LIN {X 0,Y 390.113,Z 239.893,A -85,B 0,C 180,E1 -11673.23,E2 -11673.23} C_VEL
LIN {X 0,Y 390.106,Z 239.893,A -85,B 0,C 180,E1 -11676.749,E2 -11676.749} C_VEL
LIN {X 0,Y 390.103,Z 239.89,A -85,B 0,C 180,E1 -11679.981,E2 -11679.981} C_VEL
LIN {X 0,Y 390.136,Z 239.889,A -85,B 0,C 180,E1 -11683.247,E2 -11683.247} C_VEL
LIN {X 0,Y 390.192,Z 239.881,A -85,B 0,C 180,E1 -11686.56,E2 -11686.56} C_VEL
LIN {X 0,Y 390.202,Z 239.882,A -85,B 0,C 180,E1 -11690.67,E2 -11690.67} C_VEL
LIN {X 0,Y 390.316,Z 239.868,A -85,B 0,C 180,E1 -11692.757,E2 -11692.757} C_VEL
LIN {X 0,Y 390.225,Z 239.879,A -85,B 0,C 180,E1 -11694.832,E2 -11694.832} C_VEL
LIN {X 0,Y 390.417,Z 239.853,A -85,B 0,C 180,E1 -11697.935,E2 -11697.935} C_VEL
LIN {X 0,Y 390.548,Z 239.838,A -85,B 0,C 180,E1 -11699.998,E2 -11699.998} C_VEL
LIN {X 0,Y 390.31,Z 239.868,A -85,B 0,C 180,E1 -11703.095,E2 -11703.095} C_VEL
LIN {X 0,Y 390.304,Z 239.868,A -85,B 0,C 180,E1 -11706.648,E2 -11706.648} C_VEL
LIN {X 0,Y 390.307,Z 239.869,A -85,B 0,C 180,E1 -11708.28,E2 -11708.28} C_VEL
LIN {X 0,Y 390.044,Z 239.907,A -85,B 0,C 180,E1 -11711.43,E2 -11711.43} C_VEL
LIN {X 0,Y 389.974,Z 239.918,A -85,B 0,C 180,E1 -11712.488,E2 -11712.488} C_VEL
LIN {X 0,Y 389.81,Z 242.6,A -85,B 0,C 180,E1 -11715.688,E2 -11715.688} C_VEL
LIN {X 0,Y 389.67,Z 245.504,A -85,B 0,C 180,E1 -11718.942,E2 -11718.942} C_VEL
LIN {X 0,Y 389.507,Z 248.517,A -85,B 0,C 180,E1 -11722.264,E2 -11722.264} C_VEL
LIN {X 0,Y 389.405,Z 251.667,A -85,B 0,C 180,E1 -11725.665,E2 -11725.665} C_VEL
LIN {X 0,Y 389.324,Z 254.422,A -85,B 0,C 180,E1 -11728.43,E2 -11728.43} C_VEL
LIN {X 0,Y 393.252,Z 268.11,A -85,B 0,C 180,E1 -11729.178,E2 -11729.178} C_VEL
LIN {X 0,Y 395.406,Z 278.173,A -85,B 0,C 180,E1 -11729.844,E2 -11729.844} C_VEL
LIN {X 0,Y 394.652,Z 289.978,A -85,B 0,C 180,E1 -11730.645,E2 -11730.645} C_VEL
LIN {X 0,Y 393.838,Z 300.965,A -85,B 0,C 180,E1 -11731.611,E2 -11731.611} C_VEL
LIN {X 0,Y 392.925,Z 311.66,A -85,B 0,C 180,E1 -11732.792,E2 -11732.792} C_VEL
LIN {X 0,Y 392.087,Z 321.028,A -85,B 0,C 180,E1 -11734.072,E2 -11734.072} C_VEL
LIN {X 0,Y 391.283,Z 329.692,A -85,B 0,C 180,E1 -11735.54,E2 -11735.54} C_VEL
LIN {X 0,Y 390.59,Z 336.658,A -85,B 0,C 180,E1 -11736.997,E2 -11736.997} C_VEL
LIN {X 0,Y 389.928,Z 343.417,A -85,B 0,C 180,E1 -11738.777,E2 -11738.777} C_VEL
LIN {X 0,Y 389.469,Z 348.432,A -85,B 0,C 180,E1 -11740.51,E2 -11740.51} C_VEL
LIN {X 0,Y 389.146,Z 352.053,A -85,B 0,C 180,E1 -11742.23,E2 -11742.23} C_VEL
LIN {X 0,Y 388.911,Z 354.23,A -85,B 0,C 180,E1 -11743.712,E2 -11743.712} C_VEL
LIN {X 0,Y 388.776,Z 355.525,A -85,B 0,C 180,E1 -11745.171,E2 -11745.171} C_VEL
LIN {X 0,Y 388.69,Z 356.014,A -85,B 0,C 180,E1 -11746.601,E2 -11746.601} C_VEL
LIN {X 0,Y 388.695,Z 355.772,A -85,B 0,C 180,E1 -11748.011,E2 -11748.011} C_VEL
LIN {X 0,Y 388.784,Z 354.819,A -85,B 0,C 180,E1 -11749.402,E2 -11749.402} C_VEL
LIN {X 0,Y 388.923,Z 352.818,A -85,B 0,C 180,E1 -11750.985,E2 -11750.985} C_VEL
LIN {X 0,Y 389.183,Z 349.734,A -85,B 0,C 180,E1 -11752.61,E2 -11752.61} C_VEL
LIN {X 0,Y 389.539,Z 345.387,A -85,B 0,C 180,E1 -11754.276,E2 -11754.276} C_VEL
LIN {X 0,Y 390.009,Z 339.3,A -85,B 0,C 180,E1 -11756.04,E2 -11756.04} C_VEL
LIN {X 0,Y 390.678,Z 331.897,A -85,B 0,C 180,E1 -11757.72,E2 -11757.72} C_VEL
LIN {X 0,Y 391.288,Z 324.452,A -85,B 0,C 180,E1 -11759.083,E2 -11759.083} C_VEL
LIN {X 0,Y 392.091,Z 315.125,A -85,B 0,C 180,E1 -11760.468,E2 -11760.468} C_VEL
LIN {X 0,Y 392.899,Z 304.851,A -85,B 0,C 180,E1 -11761.705,E2 -11761.705} C_VEL
LIN {X 0,Y 393.743,Z 293.832,A -85,B 0,C 180,E1 -11762.77,E2 -11762.77} C_VEL
LIN {X 0,Y 394.509,Z 281.481,A -85,B 0,C 180,E1 -11763.697,E2 -11763.697} C_VEL
LIN {X 0,Y 394.722,Z 276.68,A -85,B 0,C 180,E1 -11763.996,E2 -11763.996} C_VEL
LIN {X 0,Y 392.619,Z 266.1,A -85,B 0,C 180,E1 -11764.653,E2 -11764.653} C_VEL
LIN {X 0,Y 389.265,Z 253.104,A -85,B 0,C 180,E1 -11765.297,E2 -11765.297} C_VEL
LIN {X 0,Y 389.144,Z 252.388,A -85,B 0,C 180,E1 -11765.356,E2 -11765.356} C_VEL
LIN {X 0,Y 389.162,Z 248.817,A -85,B 0,C 180,E1 -11768.828,E2 -11768.828} C_VEL
LIN {X 0,Y 389.251,Z 245.495,A -85,B 0,C 180,E1 -11772.126,E2 -11772.126} C_VEL
LIN {X 0,Y 389.366,Z 242.289,A -85,B 0,C 180,E1 -11775.363,E2 -11775.363} C_VEL
LIN {X 0,Y 389.493,Z 240.191,A -85,B 0,C 180,E1 -11777.495,E2 -11777.495} C_VEL
LIN {X 0,Y 389.903,Z 239.916,A -85,B 0,C 180,E1 -11780.665,E2 -11780.665} C_VEL
LIN {X 0,Y 390.217,Z 239.877,A -85,B 0,C 180,E1 -11782.758,E2 -11782.758} C_VEL
LIN {X 0,Y 390.211,Z 239.878,A -85,B 0,C 180,E1 -11784.834,E2 -11784.834} C_VEL
LIN {X 0,Y 390.405,Z 239.854,A -85,B 0,C 180,E1 -11787.937,E2 -11787.937} C_VEL
LIN {X 0,Y 390.536,Z 239.837,A -85,B 0,C 180,E1 -11790.001,E2 -11790.001} C_VEL
LIN {X 0,Y 390.302,Z 239.87,A -85,B 0,C 180,E1 -11793.097,E2 -11793.097} C_VEL
LIN {X 0,Y 390.316,Z 239.864,A -85,B 0,C 180,E1 -11796.203,E2 -11796.203} C_VEL
LIN {X 0,Y 390.299,Z 239.866,A -85,B 0,C 180,E1 -11798.283,E2 -11798.283} C_VEL
LIN {X 0,Y 390.163,Z 239.884,A -85,B 0,C 180,E1 -11802.484,E2 -11802.484} C_VEL
LIN {X 0,Y 390.125,Z 239.889,A -85,B 0,C 180,E1 -11805.678,E2 -11805.678} C_VEL
LIN {X 0,Y 390.123,Z 239.889,A -85,B 0,C 180,E1 -11807.504,E2 -11807.504} C_VEL
LIN {X 0,Y 389.437,Z 239.975,A -85,B 0,C 180,E1 -11808.367,E2 -11808.367} C_VEL
LIN {X 0,Y 386.571,Z 240.33,A -85,B 0,C 180,E1 -11809.768,E2 -11809.768} C_VEL
LIN {X 0,Y 384.154,Z 240.636,A -85,B 0,C 180,E1 -11810.901,E2 -11810.901} C_VEL
LIN {X 0,Y 383.115,Z 240.761,A -85,B 0,C 180,E1 -11811.776,E2 -11811.776} C_VEL
LIN {X 0,Y 383.028,Z 240.772,A -85,B 0,C 180,E1 -11812.073,E2 -11812.073} C_VEL
LIN {X 0,Y 383.041,Z 240.774,A -85,B 0,C 180,E1 -11814.962,E2 -11814.962} C_VEL
LIN {X 0,Y 383.027,Z 240.775,A -85,B 0,C 180,E1 -11818.494,E2 -11818.494} C_VEL
LIN {X 0,Y 382.997,Z 240.777,A -85,B 0,C 180,E1 -11822.151,E2 -11822.151} C_VEL
LIN {X 0,Y 383.007,Z 240.778,A -85,B 0,C 180,E1 -11824.67,E2 -11824.67} C_VEL
LIN {X 0,Y 382.993,Z 240.777,A -85,B 0,C 180,E1 -11827.906,E2 -11827.906} C_VEL
LIN {X 0,Y 383.037,Z 240.771,A -85,B 0,C 180,E1 -11831.341,E2 -11831.341} C_VEL
LIN {X 0,Y 383.061,Z 240.771,A -85,B 0,C 180,E1 -11834.317,E2 -11834.317} C_VEL
LIN {X 0,Y 383.067,Z 240.767,A -85,B 0,C 180,E1 -11837.251,E2 -11837.251} C_VEL
LIN {X 0,Y 383.015,Z 240.778,A -85,B 0,C 180,E1 -11840.414,E2 -11840.414} C_VEL
LIN {X 0,Y 383.02,Z 240.775,A -85,B 0,C 180,E1 -11844.047,E2 -11844.047} C_VEL
LIN {X 0,Y 383.031,Z 240.773,A -85,B 0,C 180,E1 -11847.855,E2 -11847.855} C_VEL
LIN {X 0,Y 383.059,Z 240.769,A -85,B 0,C 180,E1 -11851.722,E2 -11851.722} C_VEL
LIN {X 0,Y 383.049,Z 240.769,A -85,B 0,C 180,E1 -11855.042,E2 -11855.042} C_VEL
LIN {X 0,Y 382.991,Z 240.779,A -85,B 0,C 180,E1 -11858.471,E2 -11858.471} C_VEL
LIN {X 0,Y 383.088,Z 240.768,A -85,B 0,C 180,E1 -11861.83,E2 -11861.83} C_VEL
LIN {X 0,Y 383.109,Z 240.761,A -85,B 0,C 180,E1 -11865.12,E2 -11865.12} C_VEL
LIN {X 0,Y 383.097,Z 240.765,A -85,B 0,C 180,E1 -11868.36,E2 -11868.36} C_VEL
LIN {X 0,Y 383.229,Z 240.751,A -85,B 0,C 180,E1 -11872.016,E2 -11872.016} C_VEL
LIN {X 0,Y 383.197,Z 240.75,A -85,B 0,C 180,E1 -11874.74,E2 -11874.74} C_VEL
LIN {X 0,Y 383.387,Z 240.731,A -85,B 0,C 180,E1 -11877.901,E2 -11877.901} C_VEL
LIN {X 0,Y 383.52,Z 240.714,A -85,B 0,C 180,E1 -11880.002,E2 -11880.002} C_VEL
LIN {X 0,Y 383.247,Z 240.746,A -85,B 0,C 180,E1 -11883.155,E2 -11883.155} C_VEL
LIN {X 0,Y 383.259,Z 240.743,A -85,B 0,C 180,E1 -11886.318,E2 -11886.318} C_VEL
LIN {X 0,Y 383.147,Z 240.761,A -85,B 0,C 180,E1 -11889.504,E2 -11889.504} C_VEL
LIN {X 0,Y 383.13,Z 240.763,A -85,B 0,C 180,E1 -11893.538,E2 -11893.538} C_VEL
LIN {X 0,Y 383.101,Z 240.767,A -85,B 0,C 180,E1 -11897.456,E2 -11897.456} C_VEL
LIN {X 0,Y 383.035,Z 240.771,A -85,B 0,C 180,E1 -11900.648,E2 -11900.648} C_VEL
LIN {X 0,Y 383.038,Z 240.772,A -85,B 0,C 180,E1 -11903.809,E2 -11903.809} C_VEL
LIN {X 0,Y 383.085,Z 240.765,A -85,B 0,C 180,E1 -11906.124,E2 -11906.124} C_VEL
LIN {X 0,Y 382.998,Z 240.777,A -85,B 0,C 180,E1 -11909.701,E2 -11909.701} C_VEL
LIN {X 0,Y 383.01,Z 240.777,A -85,B 0,C 180,E1 -11913.402,E2 -11913.402} C_VEL
LIN {X 0,Y 383.038,Z 240.77,A -85,B 0,C 180,E1 -11916.165,E2 -11916.165} C_VEL
LIN {X 0,Y 383.015,Z 240.775,A -85,B 0,C 180,E1 -11919.959,E2 -11919.959} C_VEL
LIN {X 0,Y 383.013,Z 240.774,A -85,B 0,C 180,E1 -11922.779,E2 -11922.779} C_VEL
LIN {X 0,Y 383.031,Z 240.897,A -85,B 0,C 180,E1 -11925.041,E2 -11925.041} C_VEL
LIN {X 0,Y 384.242,Z 247.351,A -85,B 0,C 180,E1 -11928.817,E2 -11928.817} C_VEL
LIN {X 0,Y 385.155,Z 252.557,A -85,B 0,C 180,E1 -11931.688,E2 -11931.688} C_VEL
LIN {X 0,Y 385.511,Z 255.721,A -85,B 0,C 180,E1 -11933.336,E2 -11933.336} C_VEL
LIN {X 0,Y 385.213,Z 260.202,A -85,B 0,C 180,E1 -11935.557,E2 -11935.557} C_VEL
LIN {X 0,Y 384.634,Z 266.612,A -85,B 0,C 180,E1 -11938.617,E2 -11938.617} C_VEL
LIN {X 0,Y 383.929,Z 274.316,A -85,B 0,C 180,E1 -11942.173,E2 -11942.173} C_VEL
LIN {X 0,Y 383.292,Z 282.084,A -85,B 0,C 180,E1 -11945.634,E2 -11945.634} C_VEL
LIN {X 0,Y 382.82,Z 289.815,A -85,B 0,C 180,E1 -11949.023,E2 -11949.023} C_VEL
LIN {X 0,Y 382.55,Z 294.774,A -85,B 0,C 180,E1 -11951.122,E2 -11951.122} C_VEL
LIN {X 0,Y 384.801,Z 308.327,A -85,B 0,C 180,E1 -11951.674,E2 -11951.674} C_VEL
LIN {X 0,Y 386.56,Z 321.861,A -85,B 0,C 180,E1 -11952.444,E2 -11952.444} C_VEL
LIN {X 0,Y 387.251,Z 328.496,A -85,B 0,C 180,E1 -11952.905,E2 -11952.905} C_VEL
LIN {X 0,Y 386.322,Z 339.658,A -85,B 0,C 180,E1 -11953.757,E2 -11953.757} C_VEL
LIN {X 0,Y 385.409,Z 350.422,A -85,B 0,C 180,E1 -11954.803,E2 -11954.803} C_VEL
LIN {X 0,Y 384.59,Z 360.711,A -85,B 0,C 180,E1 -11956.052,E2 -11956.052} C_VEL
LIN {X 0,Y 383.652,Z 370.811,A -85,B 0,C 180,E1 -11957.57,E2 -11957.57} C_VEL
LIN {X 0,Y 382.845,Z 379.183,A -85,B 0,C 180,E1 -11959.154,E2 -11959.154} C_VEL
LIN {X 0,Y 382.337,Z 385.943,A -85,B 0,C 180,E1 -11960.744,E2 -11960.744} C_VEL
LIN {X 0,Y 381.931,Z 392.145,A -85,B 0,C 180,E1 -11962.599,E2 -11962.599} C_VEL
LIN {X 0,Y 381.734,Z 396.089,A -85,B 0,C 180,E1 -11964.152,E2 -11964.152} C_VEL
LIN {X 0,Y 381.658,Z 399.137,A -85,B 0,C 180,E1 -11965.775,E2 -11965.775} C_VEL
LIN {X 0,Y 381.612,Z 400.554,A -85,B 0,C 180,E1 -11966.832,E2 -11966.832} C_VEL
LIN {X 0,Y 381.704,Z 401.564,A -85,B 0,C 180,E1 -11967.889,E2 -11967.889} C_VEL
LIN {X 0,Y 381.67,Z 402.17,A -85,B 0,C 180,E1 -11968.944,E2 -11968.944} C_VEL
LIN {X 0,Y 381.665,Z 402.382,A -85,B 0,C 180,E1 -11969.999,E2 -11969.999} C_VEL
LIN {X 0,Y 381.67,Z 402.156,A -85,B 0,C 180,E1 -11971.055,E2 -11971.055} C_VEL
LIN {X 0,Y 381.706,Z 401.528,A -85,B 0,C 180,E1 -11972.11,E2 -11972.11} C_VEL
LIN {X 0,Y 381.66,Z 399.069,A -85,B 0,C 180,E1 -11974.223,E2 -11974.223} C_VEL
LIN {X 0,Y 381.734,Z 395.99,A -85,B 0,C 180,E1 -11975.849,E2 -11975.849} C_VEL
LIN {X 0,Y 381.931,Z 392.026,A -85,B 0,C 180,E1 -11977.4,E2 -11977.4} C_VEL
LIN {X 0,Y 382.335,Z 385.829,A -85,B 0,C 180,E1 -11979.255,E2 -11979.255} C_VEL
LIN {X 0,Y 382.836,Z 379.075,A -85,B 0,C 180,E1 -11980.845,E2 -11980.845} C_VEL
LIN {X 0,Y 383.639,Z 370.727,A -85,B 0,C 180,E1 -11982.43,E2 -11982.43} C_VEL
LIN {X 0,Y 384.429,Z 362.201,A -85,B 0,C 180,E1 -11983.748,E2 -11983.748} C_VEL
LIN {X 0,Y 385.287,Z 351.704,A -85,B 0,C 180,E1 -11985.065,E2 -11985.065} C_VEL
LIN {X 0,Y 386.34,Z 339.954,A -85,B 0,C 180,E1 -11986.241,E2 -11986.241} C_VEL
LIN {X 0,Y 387.266,Z 328.929,A -85,B 0,C 180,E1 -11987.107,E2 -11987.107} C_VEL
LIN {X 0,Y 386.277,Z 318.781,A -85,B 0,C 180,E1 -11987.814,E2 -11987.814} C_VEL
LIN {X 0,Y 384.571,Z 305.331,A -85,B 0,C 180,E1 -11988.552,E2 -11988.552} C_VEL
LIN {X 0,Y 382.544,Z 293.606,A -85,B 0,C 180,E1 -11989.066,E2 -11989.066} C_VEL
LIN {X 0,Y 382.95,Z 285.205,A -85,B 0,C 180,E1 -11992.668,E2 -11992.668} C_VEL
LIN {X 0,Y 383.5,Z 277.443,A -85,B 0,C 180,E1 -11996.105,E2 -11996.105} C_VEL
LIN {X 0,Y 384.155,Z 269.858,A -85,B 0,C 180,E1 -11999.6,E2 -11999.6} C_VEL
LIN {X 0,Y 384.893,Z 262.38,A -85,B 0,C 180,E1 -12003.215,E2 -12003.215} C_VEL
LIN {X 0,Y 385.502,Z 257.518,A -85,B 0,C 180,E1 -12005.688,E2 -12005.688} C_VEL
LIN {X 0,Y 385.35,Z 253.932,A -85,B 0,C 180,E1 -12007.646,E2 -12007.646} C_VEL
LIN {X 0,Y 384.342,Z 248.124,A -85,B 0,C 180,E1 -12011.168,E2 -12011.168} C_VEL
LIN {X 0,Y 383.464,Z 243.335,A -85,B 0,C 180,E1 -12014.373,E2 -12014.373} C_VEL
LIN {X 0,Y 383.024,Z 240.775,A -85,B 0,C 180,E1 -12016.34,E2 -12016.34} C_VEL
LIN {X 0,Y 383.021,Z 240.775,A -85,B 0,C 180,E1 -12020.042,E2 -12020.042} C_VEL
LIN {X 0,Y 383.034,Z 240.776,A -85,B 0,C 180,E1 -12023.834,E2 -12023.834} C_VEL
LIN {X 0,Y 383.004,Z 240.778,A -85,B 0,C 180,E1 -12026.598,E2 -12026.598} C_VEL
LIN {X 0,Y 382.992,Z 240.779,A -85,B 0,C 180,E1 -12030.299,E2 -12030.299} C_VEL
LIN {X 0,Y 383.08,Z 240.769,A -85,B 0,C 180,E1 -12034.019,E2 -12034.019} C_VEL
LIN {X 0,Y 383.008,Z 240.774,A -85,B 0,C 180,E1 -12037.334,E2 -12037.334} C_VEL
LIN {X 0,Y 383.059,Z 240.771,A -85,B 0,C 180,E1 -12040.715,E2 -12040.715} C_VEL
LIN {X 0,Y 383.079,Z 240.767,A -85,B 0,C 180,E1 -12044.025,E2 -12044.025} C_VEL
LIN {X 0,Y 383.134,Z 240.761,A -85,B 0,C 180,E1 -12047.282,E2 -12047.282} C_VEL
LIN {X 0,Y 383.149,Z 240.76,A -85,B 0,C 180,E1 -12050.496,E2 -12050.496} C_VEL
LIN {X 0,Y 383.27,Z 240.745,A -85,B 0,C 180,E1 -12052.624,E2 -12052.624} C_VEL
LIN {X 0,Y 383.197,Z 240.755,A -85,B 0,C 180,E1 -12054.737,E2 -12054.737} C_VEL
LIN {X 0,Y 383.384,Z 240.729,A -85,B 0,C 180,E1 -12057.897,E2 -12057.897} C_VEL
LIN {X 0,Y 383.517,Z 240.714,A -85,B 0,C 180,E1 -12059.998,E2 -12059.998} C_VEL
LIN {X 0,Y 383.247,Z 240.748,A -85,B 0,C 180,E1 -12063.152,E2 -12063.152} C_VEL
LIN {X 0,Y 383.264,Z 240.746,A -85,B 0,C 180,E1 -12066.642,E2 -12066.642} C_VEL
LIN {X 0,Y 383.253,Z 240.748,A -85,B 0,C 180,E1 -12068.434,E2 -12068.434} C_VEL
LIN {X 0,Y 382.974,Z 240.789,A -85,B 0,C 180,E1 -12071.644,E2 -12071.644} C_VEL
LIN {X 0,Y 382.931,Z 241.115,A -85,B 0,C 180,E1 -12072.721,E2 -12072.721} C_VEL
LIN {X 0,Y 382.768,Z 243.881,A -85,B 0,C 180,E1 -12075.985,E2 -12075.985} C_VEL
LIN {X 0,Y 382.603,Z 246.794,A -85,B 0,C 180,E1 -12079.305,E2 -12079.305} C_VEL
LIN {X 0,Y 382.447,Z 250.316,A -85,B 0,C 180,E1 -12083.248,E2 -12083.248} C_VEL
LIN {X 0,Y 382.322,Z 253.025,A -85,B 0,C 180,E1 -12086.177,E2 -12086.177} C_VEL
LIN {X 0,Y 382.267,Z 254.753,A -85,B 0,C 180,E1 -12088.035,E2 -12088.035} C_VEL
LIN {X 0,Y 386.188,Z 268.214,A -85,B 0,C 180,E1 -12088.793,E2 -12088.793} C_VEL
LIN {X 0,Y 388.609,Z 278.77,A -85,B 0,C 180,E1 -12089.52,E2 -12089.52} C_VEL
LIN {X 0,Y 387.911,Z 290.239,A -85,B 0,C 180,E1 -12090.316,E2 -12090.316} C_VEL
LIN {X 0,Y 387.072,Z 301.265,A -85,B 0,C 180,E1 -12091.297,E2 -12091.297} C_VEL
LIN {X 0,Y 386.124,Z 311.791,A -85,B 0,C 180,E1 -12092.473,E2 -12092.473} C_VEL
LIN {X 0,Y 385.214,Z 321.436,A -85,B 0,C 180,E1 -12093.808,E2 -12093.808} C_VEL
LIN {X 0,Y 384.396,Z 329.716,A -85,B 0,C 180,E1 -12095.223,E2 -12095.223} C_VEL
LIN {X 0,Y 383.562,Z 337.849,A -85,B 0,C 180,E1 -12096.97,E2 -12096.97} C_VEL
LIN {X 0,Y 382.917,Z 343.879,A -85,B 0,C 180,E1 -12098.608,E2 -12098.608} C_VEL
LIN {X 0,Y 382.5,Z 347.977,A -85,B 0,C 180,E1 -12100.019,E2 -12100.019} C_VEL
LIN {X 0,Y 382.214,Z 351.232,A -85,B 0,C 180,E1 -12101.446,E2 -12101.446} C_VEL
LIN {X 0,Y 381.956,Z 353.723,A -85,B 0,C 180,E1 -12102.903,E2 -12102.903} C_VEL
LIN {X 0,Y 381.752,Z 355.436,A -85,B 0,C 180,E1 -12104.39,E2 -12104.39} C_VEL
LIN {X 0,Y 381.628,Z 356.323,A -85,B 0,C 180,E1 -12105.904,E2 -12105.904} C_VEL
LIN {X 0,Y 381.605,Z 356.385,A -85,B 0,C 180,E1 -12107.446,E2 -12107.446} C_VEL
LIN {X 0,Y 381.651,Z 355.576,A -85,B 0,C 180,E1 -12109.022,E2 -12109.022} C_VEL
LIN {X 0,Y 381.798,Z 353.82,A -85,B 0,C 180,E1 -12110.631,E2 -12110.631} C_VEL
LIN {X 0,Y 382.116,Z 350.279,A -85,B 0,C 180,E1 -12112.632,E2 -12112.632} C_VEL
LIN {X 0,Y 382.572,Z 345.011,A -85,B 0,C 180,E1 -12114.644,E2 -12114.644} C_VEL
LIN {X 0,Y 382.99,Z 339.839,A -85,B 0,C 180,E1 -12116.151,E2 -12116.151} C_VEL
LIN {X 0,Y 383.693,Z 332.203,A -85,B 0,C 180,E1 -12117.915,E2 -12117.915} C_VEL
LIN {X 0,Y 384.477,Z 323.212,A -85,B 0,C 180,E1 -12119.546,E2 -12119.546} C_VEL
LIN {X 0,Y 385.25,Z 314.53,A -85,B 0,C 180,E1 -12120.823,E2 -12120.823} C_VEL
LIN {X 0,Y 386.09,Z 304.338,A -85,B 0,C 180,E1 -12122.049,E2 -12122.049} C_VEL
LIN {X 0,Y 386.961,Z 292.894,A -85,B 0,C 180,E1 -12123.143,E2 -12123.143} C_VEL
LIN {X 0,Y 387.698,Z 281.55,A -85,B 0,C 180,E1 -12123.995,E2 -12123.995} C_VEL
LIN {X 0,Y 387.911,Z 277.906,A -85,B 0,C 180,E1 -12124.227,E2 -12124.227} C_VEL
LIN {X 0,Y 386.165,Z 268.817,A -85,B 0,C 180,E1 -12124.824,E2 -12124.824} C_VEL
LIN {X 0,Y 383.077,Z 256.65,A -85,B 0,C 180,E1 -12125.476,E2 -12125.476} C_VEL
LIN {X 0,Y 382.066,Z 252.795,A -85,B 0,C 180,E1 -12125.66,E2 -12125.66} C_VEL
LIN {X 0,Y 382.079,Z 249.982,A -85,B 0,C 180,E1 -12128.416,E2 -12128.416} C_VEL
LIN {X 0,Y 382.183,Z 246.611,A -85,B 0,C 180,E1 -12131.784,E2 -12131.784} C_VEL
LIN {X 0,Y 382.286,Z 243.366,A -85,B 0,C 180,E1 -12135.086,E2 -12135.086} C_VEL
LIN {X 0,Y 382.434,Z 241.248,A -85,B 0,C 180,E1 -12137.261,E2 -12137.261} C_VEL
LIN {X 0,Y 382.664,Z 240.822,A -85,B 0,C 180,E1 -12139.418,E2 -12139.418} C_VEL
LIN {X 0,Y 383.156,Z 240.756,A -85,B 0,C 180,E1 -12142.624,E2 -12142.624} C_VEL
LIN {X 0,Y 383.182,Z 240.753,A -85,B 0,C 180,E1 -12144.739,E2 -12144.739} C_VEL
LIN {X 0,Y 383.372,Z 240.73,A -85,B 0,C 180,E1 -12147.899,E2 -12147.899} C_VEL
LIN {X 0,Y 383.505,Z 240.712,A -85,B 0,C 180,E1 -12150.001,E2 -12150.001} C_VEL
LIN {X 0,Y 383.238,Z 240.75,A -85,B 0,C 180,E1 -12153.154,E2 -12153.154} C_VEL
LIN {X 0,Y 383.273,Z 240.741,A -85,B 0,C 180,E1 -12156.317,E2 -12156.317} C_VEL
LIN {X 0,Y 383.245,Z 240.745,A -85,B 0,C 180,E1 -12158.437,E2 -12158.437} C_VEL
LIN {X 0,Y 383.093,Z 240.764,A -85,B 0,C 180,E1 -12161.643,E2 -12161.643} C_VEL
LIN {X 0,Y 383.097,Z 240.767,A -85,B 0,C 180,E1 -12164.883,E2 -12164.883} C_VEL
LIN {X 0,Y 383.08,Z 240.765,A -85,B 0,C 180,E1 -12168.173,E2 -12168.173} C_VEL
LIN {X 0,Y 383.056,Z 240.769,A -85,B 0,C 180,E1 -12171.528,E2 -12171.528} C_VEL
LIN {X 0,Y 383.028,Z 240.772,A -85,B 0,C 180,E1 -12172.073,E2 -12172.073} C_VEL
LIN {X 0,Y 382.371,Z 240.858,A -85,B 0,C 180,E1 -12172.95,E2 -12172.95} C_VEL
LIN {X 0,Y 379.566,Z 241.213,A -85,B 0,C 180,E1 -12174.377,E2 -12174.377} C_VEL
LIN {X 0,Y 377.168,Z 241.512,A -85,B 0,C 180,E1 -12175.529,E2 -12175.529} C_VEL
LIN {X 0,Y 376.105,Z 241.64,A -85,B 0,C 180,E1 -12176.42,E2 -12176.42} C_VEL
LIN {X 0,Y 376,Z 241.65,A -85,B 0,C 180,E1 -12176.722,E2 -12176.722} C_VEL
LIN {X 0,Y 375.952,Z 241.654,A -85,B 0,C 180,E1 -12180.314,E2 -12180.314} C_VEL
LIN {X 0,Y 375.948,Z 241.654,A -85,B 0,C 180,E1 -12184.113,E2 -12184.113} C_VEL
LIN {X 0,Y 375.944,Z 241.658,A -85,B 0,C 180,E1 -12186.743,E2 -12186.743} C_VEL
LIN {X 0,Y 375.989,Z 241.649,A -85,B 0,C 180,E1 -12189.975,E2 -12189.975} C_VEL
LIN {X 0,Y 375.99,Z 241.648,A -85,B 0,C 180,E1 -12193.758,E2 -12193.758} C_VEL
LIN {X 0,Y 375.991,Z 241.651,A -85,B 0,C 180,E1 -12196.802,E2 -12196.802} C_VEL
LIN {X 0,Y 375.992,Z 241.65,A -85,B 0,C 180,E1 -12200.029,E2 -12200.029} C_VEL
LIN {X 0,Y 375.959,Z 241.652,A -85,B 0,C 180,E1 -12203.497,E2 -12203.497} C_VEL
LIN {X 0,Y 375.957,Z 241.654,A -85,B 0,C 180,E1 -12205.891,E2 -12205.891} C_VEL
LIN {X 0,Y 375.965,Z 241.652,A -85,B 0,C 180,E1 -12209.69,E2 -12209.69} C_VEL
LIN {X 0,Y 375.999,Z 241.651,A -85,B 0,C 180,E1 -12212.144,E2 -12212.144} C_VEL
LIN {X 0,Y 376.003,Z 241.649,A -85,B 0,C 180,E1 -12214.541,E2 -12214.541} C_VEL
LIN {X 0,Y 375.961,Z 241.656,A -85,B 0,C 180,E1 -12218.048,E2 -12218.048} C_VEL
LIN {X 0,Y 376.022,Z 241.645,A -85,B 0,C 180,E1 -12221.476,E2 -12221.476} C_VEL
LIN {X 0,Y 376.058,Z 241.64,A -85,B 0,C 180,E1 -12224.835,E2 -12224.835} C_VEL
LIN {X 0,Y 376.049,Z 241.645,A -85,B 0,C 180,E1 -12228.139,E2 -12228.139} C_VEL
LIN {X 0,Y 376.201,Z 241.626,A -85,B 0,C 180,E1 -12231.941,E2 -12231.941} C_VEL
LIN {X 0,Y 376.169,Z 241.626,A -85,B 0,C 180,E1 -12234.642,E2 -12234.642} C_VEL
LIN {X 0,Y 376.353,Z 241.607,A -85,B 0,C 180,E1 -12237.861,E2 -12237.861} C_VEL
LIN {X 0,Y 376.49,Z 241.589,A -85,B 0,C 180,E1 -12240.002,E2 -12240.002} C_VEL
LIN {X 0,Y 376.185,Z 241.625,A -85,B 0,C 180,E1 -12243.215,E2 -12243.215} C_VEL
LIN {X 0,Y 376.217,Z 241.62,A -85,B 0,C 180,E1 -12246.437,E2 -12246.437} C_VEL
LIN {X 0,Y 376.117,Z 241.637,A -85,B 0,C 180,E1 -12249.683,E2 -12249.683} C_VEL
LIN {X 0,Y 376.095,Z 241.639,A -85,B 0,C 180,E1 -12253.659,E2 -12253.659} C_VEL
LIN {X 0,Y 376.049,Z 241.645,A -85,B 0,C 180,E1 -12257.608,E2 -12257.608} C_VEL
LIN {X 0,Y 375.984,Z 241.65,A -85,B 0,C 180,E1 -12260.833,E2 -12260.833} C_VEL
LIN {X 0,Y 375.998,Z 241.647,A -85,B 0,C 180,E1 -12264.283,E2 -12264.283} C_VEL
LIN {X 0,Y 376.026,Z 241.645,A -85,B 0,C 180,E1 -12266.653,E2 -12266.653} C_VEL
LIN {X 0,Y 375.971,Z 241.65,A -85,B 0,C 180,E1 -12270.314,E2 -12270.314} C_VEL
LIN {X 0,Y 375.966,Z 241.651,A -85,B 0,C 180,E1 -12274.112,E2 -12274.112} C_VEL
LIN {X 0,Y 375.96,Z 241.654,A -85,B 0,C 180,E1 -12276.742,E2 -12276.742} C_VEL
LIN {X 0,Y 375.995,Z 241.649,A -85,B 0,C 180,E1 -12279.971,E2 -12279.971} C_VEL
LIN {X 0,Y 375.937,Z 241.655,A -85,B 0,C 180,E1 -12283.767,E2 -12283.767} C_VEL
LIN {X 0,Y 376.011,Z 241.888,A -85,B 0,C 180,E1 -12284.744,E2 -12284.744} C_VEL
LIN {X 0,Y 377.095,Z 247.658,A -85,B 0,C 180,E1 -12288.203,E2 -12288.203} C_VEL
LIN {X 0,Y 378.067,Z 253.177,A -85,B 0,C 180,E1 -12291.331,E2 -12291.331} C_VEL
LIN {X 0,Y 378.513,Z 257.32,A -85,B 0,C 180,E1 -12293.547,E2 -12293.547} C_VEL
LIN {X 0,Y 378.107,Z 262.434,A -85,B 0,C 180,E1 -12296.108,E2 -12296.108} C_VEL
LIN {X 0,Y 377.503,Z 268.237,A -85,B 0,C 180,E1 -12298.915,E2 -12298.915} C_VEL
LIN {X 0,Y 376.852,Z 275.246,A -85,B 0,C 180,E1 -12302.21,E2 -12302.21} C_VEL
LIN {X 0,Y 376.21,Z 282.972,A -85,B 0,C 180,E1 -12305.733,E2 -12305.733} C_VEL
LIN {X 0,Y 375.7,Z 290.942,A -85,B 0,C 180,E1 -12309.283,E2 -12309.283} C_VEL
LIN {X 0,Y 375.51,Z 294.342,A -85,B 0,C 180,E1 -12310.775,E2 -12310.775} C_VEL
LIN {X 0,Y 377.773,Z 308.029,A -85,B 0,C 180,E1 -12311.345,E2 -12311.345} C_VEL
LIN {X 0,Y 379.393,Z 320.576,A -85,B 0,C 180,E1 -12312.068,E2 -12312.068} C_VEL
LIN {X 0,Y 380.322,Z 329.463,A -85,B 0,C 180,E1 -12312.7,E2 -12312.7} C_VEL
LIN {X 0,Y 379.218,Z 341.944,A -85,B 0,C 180,E1 -12313.721,E2 -12313.721} C_VEL
LIN {X 0,Y 378.192,Z 353.38,A -85,B 0,C 180,E1 -12314.92,E2 -12314.92} C_VEL
LIN {X 0,Y 377.306,Z 363.513,A -85,B 0,C 180,E1 -12316.261,E2 -12316.261} C_VEL
LIN {X 0,Y 376.379,Z 373.302,A -85,B 0,C 180,E1 -12317.873,E2 -12317.873} C_VEL
LIN {X 0,Y 375.665,Z 381.144,A -85,B 0,C 180,E1 -12319.49,E2 -12319.49} C_VEL
LIN {X 0,Y 375.081,Z 388.335,A -85,B 0,C 180,E1 -12321.378,E2 -12321.378} C_VEL
LIN {X 0,Y 374.772,Z 393.133,A -85,B 0,C 180,E1 -12322.998,E2 -12322.998} C_VEL
LIN {X 0,Y 374.65,Z 396.805,A -85,B 0,C 180,E1 -12324.618,E2 -12324.618} C_VEL
LIN {X 0,Y 374.588,Z 398.698,A -85,B 0,C 180,E1 -12325.695,E2 -12325.695} C_VEL
LIN {X 0,Y 374.523,Z 400.121,A -85,B 0,C 180,E1 -12326.772,E2 -12326.772} C_VEL
LIN {X 0,Y 374.606,Z 401.133,A -85,B 0,C 180,E1 -12327.849,E2 -12327.849} C_VEL
LIN {X 0,Y 374.605,Z 401.744,A -85,B 0,C 180,E1 -12328.924,E2 -12328.924} C_VEL
LIN {X 0,Y 374.597,Z 401.959,A -85,B 0,C 180,E1 -12329.999,E2 -12329.999} C_VEL
LIN {X 0,Y 374.605,Z 401.738,A -85,B 0,C 180,E1 -12331.074,E2 -12331.074} C_VEL
LIN {X 0,Y 374.609,Z 401.109,A -85,B 0,C 180,E1 -12332.15,E2 -12332.15} C_VEL
LIN {X 0,Y 374.589,Z 398.656,A -85,B 0,C 180,E1 -12334.303,E2 -12334.303} C_VEL
LIN {X 0,Y 374.702,Z 394.965,A -85,B 0,C 180,E1 -12336.229,E2 -12336.229} C_VEL
LIN {X 0,Y 374.947,Z 390.011,A -85,B 0,C 180,E1 -12338.081,E2 -12338.081} C_VEL
LIN {X 0,Y 375.395,Z 384.415,A -85,B 0,C 180,E1 -12339.7,E2 -12339.7} C_VEL
LIN {X 0,Y 375.951,Z 377.444,A -85,B 0,C 180,E1 -12341.319,E2 -12341.319} C_VEL
LIN {X 0,Y 376.846,Z 368.778,A -85,B 0,C 180,E1 -12342.931,E2 -12342.931} C_VEL
LIN {X 0,Y 377.729,Z 359.513,A -85,B 0,C 180,E1 -12344.329,E2 -12344.329} C_VEL
LIN {X 0,Y 378.62,Z 349.068,A -85,B 0,C 180,E1 -12345.613,E2 -12345.613} C_VEL
LIN {X 0,Y 379.677,Z 338.251,A -85,B 0,C 180,E1 -12346.672,E2 -12346.672} C_VEL
LIN {X 0,Y 380.431,Z 328.882,A -85,B 0,C 180,E1 -12347.418,E2 -12347.418} C_VEL
LIN {X 0,Y 379.093,Z 316.098,A -85,B 0,C 180,E1 -12348.313,E2 -12348.313} C_VEL
LIN {X 0,Y 377.288,Z 302.907,A -85,B 0,C 180,E1 -12349.03,E2 -12349.03} C_VEL
LIN {X 0,Y 375.502,Z 293.117,A -85,B 0,C 180,E1 -12349.473,E2 -12349.473} C_VEL
LIN {X 0,Y 375.964,Z 284.865,A -85,B 0,C 180,E1 -12353.113,E2 -12353.113} C_VEL
LIN {X 0,Y 376.528,Z 277.186,A -85,B 0,C 180,E1 -12356.612,E2 -12356.612} C_VEL
LIN {X 0,Y 377.258,Z 269.596,A -85,B 0,C 180,E1 -12360.197,E2 -12360.197} C_VEL
LIN {X 0,Y 378.063,Z 262.177,A -85,B 0,C 180,E1 -12363.895,E2 -12363.895} C_VEL
LIN {X 0,Y 378.526,Z 257.339,A -85,B 0,C 180,E1 -12366.45,E2 -12366.45} C_VEL
LIN {X 0,Y 378.112,Z 253.551,A -85,B 0,C 180,E1 -12368.677,E2 -12368.677} C_VEL
LIN {X 0,Y 377.121,Z 248.122,A -85,B 0,C 180,E1 -12372.135,E2 -12372.135} C_VEL
LIN {X 0,Y 376.36,Z 243.746,A -85,B 0,C 180,E1 -12375.201,E2 -12375.201} C_VEL
LIN {X 0,Y 375.977,Z 241.653,A -85,B 0,C 180,E1 -12376.888,E2 -12376.888} C_VEL
LIN {X 0,Y 375.97,Z 241.655,A -85,B 0,C 180,E1 -12380.537,E2 -12380.537} C_VEL
LIN {X 0,Y 375.966,Z 241.654,A -85,B 0,C 180,E1 -12383.494,E2 -12383.494} C_VEL
LIN {X 0,Y 375.961,Z 241.658,A -85,B 0,C 180,E1 -12385.887,E2 -12385.887} C_VEL
LIN {X 0,Y 375.965,Z 241.655,A -85,B 0,C 180,E1 -12389.686,E2 -12389.686} C_VEL
LIN {X 0,Y 376.019,Z 241.648,A -85,B 0,C 180,E1 -12393.346,E2 -12393.346} C_VEL
LIN {X 0,Y 375.996,Z 241.65,A -85,B 0,C 180,E1 -12396.887,E2 -12396.887} C_VEL
LIN {X 0,Y 375.997,Z 241.648,A -85,B 0,C 180,E1 -12400.338,E2 -12400.338} C_VEL
LIN {X 0,Y 376.027,Z 241.646,A -85,B 0,C 180,E1 -12403.717,E2 -12403.717} C_VEL
LIN {X 0,Y 376.101,Z 241.635,A -85,B 0,C 180,E1 -12407.04,E2 -12407.04} C_VEL
LIN {X 0,Y 376.116,Z 241.636,A -85,B 0,C 180,E1 -12410.317,E2 -12410.317} C_VEL
LIN {X 0,Y 376.227,Z 241.622,A -85,B 0,C 180,E1 -12412.485,E2 -12412.485} C_VEL
LIN {X 0,Y 376.169,Z 241.63,A -85,B 0,C 180,E1 -12414.638,E2 -12414.638} C_VEL
LIN {X 0,Y 376.35,Z 241.604,A -85,B 0,C 180,E1 -12417.858,E2 -12417.858} C_VEL
LIN {X 0,Y 376.487,Z 241.589,A -85,B 0,C 180,E1 -12419.998,E2 -12419.998} C_VEL
LIN {X 0,Y 376.185,Z 241.628,A -85,B 0,C 180,E1 -12423.211,E2 -12423.211} C_VEL
LIN {X 0,Y 376.228,Z 241.622,A -85,B 0,C 180,E1 -12426.634,E2 -12426.634} C_VEL
LIN {X 0,Y 376.197,Z 241.627,A -85,B 0,C 180,E1 -12428.593,E2 -12428.593} C_VEL
LIN {X 0,Y 375.901,Z 241.671,A -85,B 0,C 180,E1 -12431.866,E2 -12431.866} C_VEL
LIN {X 0,Y 375.842,Z 243.287,A -85,B 0,C 180,E1 -12434.067,E2 -12434.067} C_VEL
LIN {X 0,Y 375.693,Z 246.147,A -85,B 0,C 180,E1 -12437.44,E2 -12437.44} C_VEL
LIN {X 0,Y 375.482,Z 249.097,A -85,B 0,C 180,E1 -12440.83,E2 -12440.83} C_VEL
LIN {X 0,Y 375.351,Z 252.213,A -85,B 0,C 180,E1 -12444.323,E2 -12444.323} C_VEL
LIN {X 0,Y 375.237,Z 255.227,A -85,B 0,C 180,E1 -12447.614,E2 -12447.614} C_VEL
LIN {X 0,Y 379.521,Z 269.824,A -85,B 0,C 180,E1 -12448.487,E2 -12448.487} C_VEL
LIN {X 0,Y 381.857,Z 279.815,A -85,B 0,C 180,E1 -12449.208,E2 -12449.208} C_VEL
LIN {X 0,Y 381.178,Z 290.907,A -85,B 0,C 180,E1 -12450.001,E2 -12450.001} C_VEL
LIN {X 0,Y 380.28,Z 301.946,A -85,B 0,C 180,E1 -12451.007,E2 -12451.007} C_VEL
LIN {X 0,Y 379.238,Z 313.002,A -85,B 0,C 180,E1 -12452.278,E2 -12452.278} C_VEL
LIN {X 0,Y 378.232,Z 323.019,A -85,B 0,C 180,E1 -12453.721,E2 -12453.721} C_VEL
LIN {X 0,Y 377.361,Z 331.553,A -85,B 0,C 180,E1 -12455.261,E2 -12455.261} C_VEL
LIN {X 0,Y 376.495,Z 339.327,A -85,B 0,C 180,E1 -12457.011,E2 -12457.011} C_VEL
LIN {X 0,Y 375.767,Z 345.609,A -85,B 0,C 180,E1 -12458.845,E2 -12458.845} C_VEL
LIN {X 0,Y 375.395,Z 349.654,A -85,B 0,C 180,E1 -12460.369,E2 -12460.369} C_VEL
LIN {X 0,Y 374.981,Z 353.618,A -85,B 0,C 180,E1 -12462.429,E2 -12462.429} C_VEL
LIN {X 0,Y 374.673,Z 356.039,A -85,B 0,C 180,E1 -12464.539,E2 -12464.539} C_VEL
LIN {X 0,Y 374.534,Z 356.824,A -85,B 0,C 180,E1 -12466.03,E2 -12466.03} C_VEL
LIN {X 0,Y 374.517,Z 356.805,A -85,B 0,C 180,E1 -12467.504,E2 -12467.504} C_VEL
LIN {X 0,Y 374.57,Z 356.072,A -85,B 0,C 180,E1 -12468.952,E2 -12468.952} C_VEL
LIN {X 0,Y 374.704,Z 354.656,A -85,B 0,C 180,E1 -12470.38,E2 -12470.38} C_VEL
LIN {X 0,Y 375.034,Z 351.032,A -85,B 0,C 180,E1 -12472.55,E2 -12472.55} C_VEL
LIN {X 0,Y 375.351,Z 347.362,A -85,B 0,C 180,E1 -12474.086,E2 -12474.086} C_VEL
LIN {X 0,Y 375.847,Z 341.798,A -85,B 0,C 180,E1 -12475.878,E2 -12475.878} C_VEL
LIN {X 0,Y 376.444,Z 335.183,A -85,B 0,C 180,E1 -12477.538,E2 -12477.538} C_VEL
LIN {X 0,Y 377.25,Z 326.81,A -85,B 0,C 180,E1 -12479.205,E2 -12479.205} C_VEL
LIN {X 0,Y 378.098,Z 317.709,A -85,B 0,C 180,E1 -12480.668,E2 -12480.668} C_VEL
LIN {X 0,Y 378.933,Z 308.035,A -85,B 0,C 180,E1 -12481.926,E2 -12481.926} C_VEL
LIN {X 0,Y 379.868,Z 297.214,A -85,B 0,C 180,E1 -12483.057,E2 -12483.057} C_VEL
LIN {X 0,Y 380.679,Z 285.044,A -85,B 0,C 180,E1 -12484.068,E2 -12484.068} C_VEL
LIN {X 0,Y 381.081,Z 279.141,A -85,B 0,C 180,E1 -12484.464,E2 -12484.464} C_VEL
LIN {X 0,Y 378.693,Z 267.299,A -85,B 0,C 180,E1 -12485.246,E2 -12485.246} C_VEL
LIN {X 0,Y 375.17,Z 254.236,A -85,B 0,C 180,E1 -12485.936,E2 -12485.936} C_VEL
LIN {X 0,Y 374.995,Z 253.135,A -85,B 0,C 180,E1 -12486.041,E2 -12486.041} C_VEL
LIN {X 0,Y 375.06,Z 249.629,A -85,B 0,C 180,E1 -12489.533,E2 -12489.533} C_VEL
LIN {X 0,Y 375.195,Z 246.391,A -85,B 0,C 180,E1 -12492.797,E2 -12492.797} C_VEL
LIN {X 0,Y 375.347,Z 242.514,A -85,B 0,C 180,E1 -12496.806,E2 -12496.806} C_VEL
LIN {X 0,Y 375.452,Z 241.722,A -85,B 0,C 180,E1 -12498.118,E2 -12498.118} C_VEL
LIN {X 0,Y 376.056,Z 241.641,A -85,B 0,C 180,E1 -12502.077,E2 -12502.077} C_VEL
LIN {X 0,Y 376.152,Z 241.628,A -85,B 0,C 180,E1 -12504.64,E2 -12504.64} C_VEL
LIN {X 0,Y 376.338,Z 241.606,A -85,B 0,C 180,E1 -12507.86,E2 -12507.86} C_VEL
LIN {X 0,Y 376.475,Z 241.588,A -85,B 0,C 180,E1 -12510.001,E2 -12510.001} C_VEL
LIN {X 0,Y 376.177,Z 241.63,A -85,B 0,C 180,E1 -12513.214,E2 -12513.214} C_VEL
LIN {X 0,Y 376.232,Z 241.618,A -85,B 0,C 180,E1 -12516.436,E2 -12516.436} C_VEL
LIN {X 0,Y 376.191,Z 241.624,A -85,B 0,C 180,E1 -12518.596,E2 -12518.596} C_VEL
LIN {X 0,Y 376.044,Z 241.641,A -85,B 0,C 180,E1 -12521.864,E2 -12521.864} C_VEL
LIN {X 0,Y 376.044,Z 241.645,A -85,B 0,C 180,E1 -12525.169,E2 -12525.169} C_VEL
LIN {X 0,Y 376.017,Z 241.646,A -85,B 0,C 180,E1 -12528.527,E2 -12528.527} C_VEL
LIN {X 0,Y 376,Z 241.646,A -85,B 0,C 180,E1 -12532.065,E2 -12532.065} C_VEL
LIN {X 0,Y 375.994,Z 241.649,A -85,B 0,C 180,E1 -12535.462,E2 -12535.462} C_VEL
LIN {X 0,Y 376,Z 241.65,A -85,B 0,C 180,E1 -12536.722,E2 -12536.722} C_VEL
LIN {X 0,Y 375.282,Z 241.737,A -85,B 0,C 180,E1 -12537.616,E2 -12537.616} C_VEL
LIN {X 0,Y 372.406,Z 242.097,A -85,B 0,C 180,E1 -12539.07,E2 -12539.07} C_VEL
LIN {X 0,Y 369.997,Z 242.398,A -85,B 0,C 180,E1 -12540.245,E2 -12540.245} C_VEL
LIN {X 0,Y 368.961,Z 242.526,A -85,B 0,C 180,E1 -12541.154,E2 -12541.154} C_VEL
LIN {X 0,Y 368.873,Z 242.535,A -85,B 0,C 180,E1 -12541.461,E2 -12541.461} C_VEL
LIN {X 0,Y 368.918,Z 242.532,A -85,B 0,C 180,E1 -12545.003,E2 -12545.003} C_VEL
LIN {X 0,Y 368.903,Z 242.536,A -85,B 0,C 180,E1 -12548.643,E2 -12548.643} C_VEL
LIN {X 0,Y 368.932,Z 242.528,A -85,B 0,C 180,E1 -12552.022,E2 -12552.022} C_VEL
LIN {X 0,Y 368.982,Z 242.521,A -85,B 0,C 180,E1 -12555.195,E2 -12555.195} C_VEL
LIN {X 0,Y 368.933,Z 242.53,A -85,B 0,C 180,E1 -12558.188,E2 -12558.188} C_VEL
LIN {X 0,Y 368.906,Z 242.53,A -85,B 0,C 180,E1 -12561.361,E2 -12561.361} C_VEL
LIN {X 0,Y 368.931,Z 242.528,A -85,B 0,C 180,E1 -12565.149,E2 -12565.149} C_VEL
LIN {X 0,Y 368.924,Z 242.528,A -85,B 0,C 180,E1 -12569.049,E2 -12569.049} C_VEL
LIN {X 0,Y 368.982,Z 242.522,A -85,B 0,C 180,E1 -12571.567,E2 -12571.567} C_VEL
LIN {X 0,Y 368.954,Z 242.524,A -85,B 0,C 180,E1 -12575.227,E2 -12575.227} C_VEL
LIN {X 0,Y 368.935,Z 242.526,A -85,B 0,C 180,E1 -12578.975,E2 -12578.975} C_VEL
LIN {X 0,Y 368.989,Z 242.524,A -85,B 0,C 180,E1 -12582.259,E2 -12582.259} C_VEL
LIN {X 0,Y 369.037,Z 242.518,A -85,B 0,C 180,E1 -12586.23,E2 -12586.23} C_VEL
LIN {X 0,Y 369.064,Z 242.515,A -85,B 0,C 180,E1 -12590.134,E2 -12590.134} C_VEL
LIN {X 0,Y 369.19,Z 242.497,A -85,B 0,C 180,E1 -12593.443,E2 -12593.443} C_VEL
LIN {X 0,Y 369.318,Z 242.484,A -85,B 0,C 180,E1 -12597.821,E2 -12597.821} C_VEL
LIN {X 0,Y 369.459,Z 242.465,A -85,B 0,C 180,E1 -12600.002,E2 -12600.002} C_VEL
LIN {X 0,Y 369.319,Z 242.481,A -85,B 0,C 180,E1 -12602.183,E2 -12602.183} C_VEL
LIN {X 0,Y 369.177,Z 242.496,A -85,B 0,C 180,E1 -12606.56,E2 -12606.56} C_VEL
LIN {X 0,Y 369.068,Z 242.514,A -85,B 0,C 180,E1 -12609.87,E2 -12609.87} C_VEL
LIN {X 0,Y 369.042,Z 242.517,A -85,B 0,C 180,E1 -12613.774,E2 -12613.774} C_VEL
LIN {X 0,Y 369.007,Z 242.521,A -85,B 0,C 180,E1 -12617.77,E2 -12617.77} C_VEL
LIN {X 0,Y 368.934,Z 242.531,A -85,B 0,C 180,E1 -12621.221,E2 -12621.221} C_VEL
LIN {X 0,Y 368.963,Z 242.524,A -85,B 0,C 180,E1 -12624.777,E2 -12624.777} C_VEL
LIN {X 0,Y 368.969,Z 242.527,A -85,B 0,C 180,E1 -12627.205,E2 -12627.205} C_VEL
LIN {X 0,Y 368.936,Z 242.53,A -85,B 0,C 180,E1 -12630.954,E2 -12630.954} C_VEL
LIN {X 0,Y 368.935,Z 242.531,A -85,B 0,C 180,E1 -12635.002,E2 -12635.002} C_VEL
LIN {X 0,Y 368.914,Z 242.533,A -85,B 0,C 180,E1 -12638.641,E2 -12638.641} C_VEL
LIN {X 0,Y 368.888,Z 242.533,A -85,B 0,C 180,E1 -12642.01,E2 -12642.01} C_VEL
LIN {X 0,Y 368.94,Z 242.7,A -85,B 0,C 180,E1 -12644.327,E2 -12644.327} C_VEL
LIN {X 0,Y 370.008,Z 248.329,A -85,B 0,C 180,E1 -12647.799,E2 -12647.799} C_VEL
LIN {X 0,Y 371.094,Z 254.419,A -85,B 0,C 180,E1 -12651.319,E2 -12651.319} C_VEL
LIN {X 0,Y 371.507,Z 258.297,A -85,B 0,C 180,E1 -12653.422,E2 -12653.422} C_VEL
LIN {X 0,Y 371.11,Z 263.275,A -85,B 0,C 180,E1 -12655.985,E2 -12655.985} C_VEL
LIN {X 0,Y 370.381,Z 269.782,A -85,B 0,C 180,E1 -12659.181,E2 -12659.181} C_VEL
LIN {X 0,Y 369.79,Z 276.17,A -85,B 0,C 180,E1 -12662.248,E2 -12662.248} C_VEL
LIN {X 0,Y 369.08,Z 284.387,A -85,B 0,C 180,E1 -12666.068,E2 -12666.068} C_VEL
LIN {X 0,Y 368.642,Z 291.02,A -85,B 0,C 180,E1 -12669.096,E2 -12669.096} C_VEL
LIN {X 0,Y 368.455,Z 293.904,A -85,B 0,C 180,E1 -12670.392,E2 -12670.392} C_VEL
LIN {X 0,Y 371.082,Z 309.892,A -85,B 0,C 180,E1 -12671.128,E2 -12671.128} C_VEL
LIN {X 0,Y 372.716,Z 323.248,A -85,B 0,C 180,E1 -12671.953,E2 -12671.953} C_VEL
LIN {X 0,Y 373.407,Z 330.115,A -85,B 0,C 180,E1 -12672.473,E2 -12672.473} C_VEL
LIN {X 0,Y 372.239,Z 342.747,A -85,B 0,C 180,E1 -12673.548,E2 -12673.548} C_VEL
LIN {X 0,Y 371.291,Z 352.798,A -85,B 0,C 180,E1 -12674.633,E2 -12674.633} C_VEL
LIN {X 0,Y 370.595,Z 361.107,A -85,B 0,C 180,E1 -12675.727,E2 -12675.727} C_VEL
LIN {X 0,Y 369.729,Z 369.775,A -85,B 0,C 180,E1 -12677.094,E2 -12677.094} C_VEL
LIN {X 0,Y 368.831,Z 378.192,A -85,B 0,C 180,E1 -12678.737,E2 -12678.737} C_VEL
LIN {X 0,Y 368.252,Z 384.982,A -85,B 0,C 180,E1 -12680.386,E2 -12680.386} C_VEL
LIN {X 0,Y 367.786,Z 391.216,A -85,B 0,C 180,E1 -12682.312,E2 -12682.312} C_VEL
LIN {X 0,Y 367.605,Z 394.92,A -85,B 0,C 180,E1 -12683.811,E2 -12683.811} C_VEL
LIN {X 0,Y 367.519,Z 398.25,A -85,B 0,C 180,E1 -12685.613,E2 -12685.613} C_VEL
LIN {X 0,Y 367.438,Z 399.683,A -85,B 0,C 180,E1 -12686.71,E2 -12686.71} C_VEL
LIN {X 0,Y 367.509,Z 400.699,A -85,B 0,C 180,E1 -12687.808,E2 -12687.808} C_VEL
LIN {X 0,Y 367.541,Z 401.315,A -85,B 0,C 180,E1 -12688.904,E2 -12688.904} C_VEL
LIN {X 0,Y 367.532,Z 401.535,A -85,B 0,C 180,E1 -12689.999,E2 -12689.999} C_VEL
LIN {X 0,Y 367.541,Z 401.322,A -85,B 0,C 180,E1 -12691.095,E2 -12691.095} C_VEL
LIN {X 0,Y 367.512,Z 400.694,A -85,B 0,C 180,E1 -12692.191,E2 -12692.191} C_VEL
LIN {X 0,Y 367.518,Z 398.248,A -85,B 0,C 180,E1 -12694.386,E2 -12694.386} C_VEL
LIN {X 0,Y 367.599,Z 394.954,A -85,B 0,C 180,E1 -12696.181,E2 -12696.181} C_VEL
LIN {X 0,Y 367.896,Z 389.622,A -85,B 0,C 180,E1 -12698.237,E2 -12698.237} C_VEL
LIN {X 0,Y 368.43,Z 383.01,A -85,B 0,C 180,E1 -12700.162,E2 -12700.162} C_VEL
LIN {X 0,Y 369.079,Z 375.779,A -85,B 0,C 180,E1 -12701.811,E2 -12701.811} C_VEL
LIN {X 0,Y 370.072,Z 366.822,A -85,B 0,C 180,E1 -12703.452,E2 -12703.452} C_VEL
LIN {X 0,Y 370.918,Z 357.655,A -85,B 0,C 180,E1 -12704.821,E2 -12704.821} C_VEL
LIN {X 0,Y 371.885,Z 347.602,A -85,B 0,C 180,E1 -12706.044,E2 -12706.044} C_VEL
LIN {X 0,Y 373.019,Z 336.494,A -85,B 0,C 180,E1 -12707.12,E2 -12707.12} C_VEL
LIN {X 0,Y 373.548,Z 328.803,A -85,B 0,C 180,E1 -12707.744,E2 -12707.744} C_VEL
LIN {X 0,Y 372.227,Z 316.219,A -85,B 0,C 180,E1 -12708.657,E2 -12708.657} C_VEL
LIN {X 0,Y 370.33,Z 302.518,A -85,B 0,C 180,E1 -12709.431,E2 -12709.431} C_VEL
LIN {X 0,Y 368.476,Z 292.675,A -85,B 0,C 180,E1 -12709.878,E2 -12709.878} C_VEL
LIN {X 0,Y 369.012,Z 283.812,A -85,B 0,C 180,E1 -12713.908,E2 -12713.908} C_VEL
LIN {X 0,Y 369.703,Z 275.638,A -85,B 0,C 180,E1 -12717.757,E2 -12717.757} C_VEL
LIN {X 0,Y 370.324,Z 269.395,A -85,B 0,C 180,E1 -12720.823,E2 -12720.823} C_VEL
LIN {X 0,Y 371.235,Z 262.048,A -85,B 0,C 180,E1 -12724.606,E2 -12724.606} C_VEL
LIN {X 0,Y 371.547,Z 258.44,A -85,B 0,C 180,E1 -12726.571,E2 -12726.571} C_VEL
LIN {X 0,Y 371.036,Z 254.3,A -85,B 0,C 180,E1 -12729.048,E2 -12729.048} C_VEL
LIN {X 0,Y 370.159,Z 249.467,A -85,B 0,C 180,E1 -12732.227,E2 -12732.227} C_VEL
LIN {X 0,Y 369.434,Z 245.237,A -85,B 0,C 180,E1 -12735.259,E2 -12735.259} C_VEL
LIN {X 0,Y 368.954,Z 242.527,A -85,B 0,C 180,E1 -12737.567,E2 -12737.567} C_VEL
LIN {X 0,Y 368.91,Z 242.535,A -85,B 0,C 180,E1 -12741.046,E2 -12741.046} C_VEL
LIN {X 0,Y 368.919,Z 242.534,A -85,B 0,C 180,E1 -12743.802,E2 -12743.802} C_VEL
LIN {X 0,Y 368.897,Z 242.534,A -85,B 0,C 180,E1 -12746.955,E2 -12746.955} C_VEL
LIN {X 0,Y 368.919,Z 242.532,A -85,B 0,C 180,E1 -12750.308,E2 -12750.308} C_VEL
LIN {X 0,Y 368.981,Z 242.524,A -85,B 0,C 180,E1 -12753.533,E2 -12753.533} C_VEL
LIN {X 0,Y 368.966,Z 242.527,A -85,B 0,C 180,E1 -12756.42,E2 -12756.42} C_VEL
LIN {X 0,Y 368.935,Z 242.526,A -85,B 0,C 180,E1 -12759.945,E2 -12759.945} C_VEL
LIN {X 0,Y 368.974,Z 242.526,A -85,B 0,C 180,E1 -12763.397,E2 -12763.397} C_VEL
LIN {X 0,Y 369.055,Z 242.513,A -85,B 0,C 180,E1 -12766.788,E2 -12766.788} C_VEL
LIN {X 0,Y 369.065,Z 242.515,A -85,B 0,C 180,E1 -12770.13,E2 -12770.13} C_VEL
LIN {X 0,Y 369.185,Z 242.5,A -85,B 0,C 180,E1 -12772.341,E2 -12772.341} C_VEL
LIN {X 0,Y 369.142,Z 242.505,A -85,B 0,C 180,E1 -12774.536,E2 -12774.536} C_VEL
LIN {X 0,Y 369.315,Z 242.481,A -85,B 0,C 180,E1 -12777.817,E2 -12777.817} C_VEL
LIN {X 0,Y 369.456,Z 242.465,A -85,B 0,C 180,E1 -12779.998,E2 -12779.998} C_VEL
LIN {X 0,Y 369.314,Z 242.484,A -85,B 0,C 180,E1 -12782.179,E2 -12782.179} C_VEL
LIN {X 0,Y 369.198,Z 242.498,A -85,B 0,C 180,E1 -12786.622,E2 -12786.622} C_VEL
LIN {X 0,Y 369.128,Z 242.508,A -85,B 0,C 180,E1 -12788.759,E2 -12788.759} C_VEL
LIN {X 0,Y 368.946,Z 242.535,A -85,B 0,C 180,E1 -12790.979,E2 -12790.979} C_VEL
LIN {X 0,Y 368.856,Z 242.796,A -85,B 0,C 180,E1 -12792.096,E2 -12792.096} C_VEL
LIN {X 0,Y 368.793,Z 244.587,A -85,B 0,C 180,E1 -12794.342,E2 -12794.342} C_VEL
LIN {X 0,Y 368.636,Z 247.436,A -85,B 0,C 180,E1 -12797.758,E2 -12797.758} C_VEL
LIN {X 0,Y 368.428,Z 250.426,A -85,B 0,C 180,E1 -12801.248,E2 -12801.248} C_VEL
LIN {X 0,Y 368.295,Z 253.571,A -85,B 0,C 180,E1 -12804.821,E2 -12804.821} C_VEL
LIN {X 0,Y 368.195,Z 255.693,A -85,B 0,C 180,E1 -12807.191,E2 -12807.191} C_VEL
LIN {X 0,Y 372.452,Z 269.916,A -85,B 0,C 180,E1 -12808.068,E2 -12808.068} C_VEL
LIN {X 0,Y 375.183,Z 281.337,A -85,B 0,C 180,E1 -12808.919,E2 -12808.919} C_VEL
LIN {X 0,Y 374.305,Z 293.475,A -85,B 0,C 180,E1 -12809.837,E2 -12809.837} C_VEL
LIN {X 0,Y 373.374,Z 304.055,A -85,B 0,C 180,E1 -12810.856,E2 -12810.856} C_VEL
LIN {X 0,Y 372.403,Z 313.963,A -85,B 0,C 180,E1 -12812.039,E2 -12812.039} C_VEL
LIN {X 0,Y 371.507,Z 322.402,A -85,B 0,C 180,E1 -12813.269,E2 -12813.269} C_VEL
LIN {X 0,Y 370.609,Z 330.344,A -85,B 0,C 180,E1 -12814.671,E2 -12814.671} C_VEL
LIN {X 0,Y 369.889,Z 336.913,A -85,B 0,C 180,E1 -12816.084,E2 -12816.084} C_VEL
LIN {X 0,Y 369.205,Z 342.43,A -85,B 0,C 180,E1 -12817.524,E2 -12817.524} C_VEL
LIN {X 0,Y 368.665,Z 346.966,A -85,B 0,C 180,E1 -12818.98,E2 -12818.98} C_VEL
LIN {X 0,Y 368.31,Z 350.607,A -85,B 0,C 180,E1 -12820.446,E2 -12820.446} C_VEL
LIN {X 0,Y 367.995,Z 353.473,A -85,B 0,C 180,E1 -12821.943,E2 -12821.943} C_VEL
LIN {X 0,Y 367.713,Z 355.574,A -85,B 0,C 180,E1 -12823.473,E2 -12823.473} C_VEL
LIN {X 0,Y 367.561,Z 356.86,A -85,B 0,C 180,E1 -12825.025,E2 -12825.025} C_VEL
LIN {X 0,Y 367.431,Z 357.332,A -85,B 0,C 180,E1 -12826.619,E2 -12826.619} C_VEL
LIN {X 0,Y 367.43,Z 356.953,A -85,B 0,C 180,E1 -12828.239,E2 -12828.239} C_VEL
LIN {X 0,Y 367.573,Z 355.67,A -85,B 0,C 180,E1 -12829.885,E2 -12829.885} C_VEL
LIN {X 0,Y 367.813,Z 353.396,A -85,B 0,C 180,E1 -12831.57,E2 -12831.57} C_VEL
LIN {X 0,Y 368.112,Z 349.982,A -85,B 0,C 180,E1 -12833.304,E2 -12833.304} C_VEL
LIN {X 0,Y 368.574,Z 345.165,A -85,B 0,C 180,E1 -12835.108,E2 -12835.108} C_VEL
LIN {X 0,Y 369.125,Z 338.962,A -85,B 0,C 180,E1 -12836.898,E2 -12836.898} C_VEL
LIN {X 0,Y 369.892,Z 331.505,A -85,B 0,C 180,E1 -12838.582,E2 -12838.582} C_VEL
LIN {X 0,Y 370.74,Z 322.84,A -85,B 0,C 180,E1 -12840.159,E2 -12840.159} C_VEL
LIN {X 0,Y 371.63,Z 312.787,A -85,B 0,C 180,E1 -12841.632,E2 -12841.632} C_VEL
LIN {X 0,Y 372.68,Z 301.358,A -85,B 0,C 180,E1 -12842.957,E2 -12842.957} C_VEL
LIN {X 0,Y 373.443,Z 291.197,A -85,B 0,C 180,E1 -12843.903,E2 -12843.903} C_VEL
LIN {X 0,Y 374.231,Z 280.32,A -85,B 0,C 180,E1 -12844.708,E2 -12844.708} C_VEL
LIN {X 0,Y 372.125,Z 269.659,A -85,B 0,C 180,E1 -12845.45,E2 -12845.45} C_VEL
LIN {X 0,Y 368.779,Z 256.973,A -85,B 0,C 180,E1 -12846.165,E2 -12846.165} C_VEL
LIN {X 0,Y 367.931,Z 253.558,A -85,B 0,C 180,E1 -12846.352,E2 -12846.352} C_VEL
LIN {X 0,Y 368.02,Z 250.025,A -85,B 0,C 180,E1 -12849.896,E2 -12849.896} C_VEL
LIN {X 0,Y 368.143,Z 246.649,A -85,B 0,C 180,E1 -12853.361,E2 -12853.361} C_VEL
LIN {X 0,Y 368.285,Z 243.382,A -85,B 0,C 180,E1 -12856.763,E2 -12856.763} C_VEL
LIN {X 0,Y 368.367,Z 242.604,A -85,B 0,C 180,E1 -12857.886,E2 -12857.886} C_VEL
LIN {X 0,Y 368.86,Z 242.541,A -85,B 0,C 180,E1 -12861.233,E2 -12861.233} C_VEL
LIN {X 0,Y 369.147,Z 242.505,A -85,B 0,C 180,E1 -12863.441,E2 -12863.441} C_VEL
LIN {X 0,Y 369.303,Z 242.482,A -85,B 0,C 180,E1 -12867.819,E2 -12867.819} C_VEL
LIN {X 0,Y 369.444,Z 242.464,A -85,B 0,C 180,E1 -12870.001,E2 -12870.001} C_VEL
LIN {X 0,Y 369.304,Z 242.481,A -85,B 0,C 180,E1 -12872.182,E2 -12872.182} C_VEL
LIN {X 0,Y 369.194,Z 242.495,A -85,B 0,C 180,E1 -12876.559,E2 -12876.559} C_VEL
LIN {X 0,Y 369.124,Z 242.506,A -85,B 0,C 180,E1 -12878.762,E2 -12878.762} C_VEL
LIN {X 0,Y 368.998,Z 242.519,A -85,B 0,C 180,E1 -12882.094,E2 -12882.094} C_VEL
LIN {X 0,Y 368.984,Z 242.523,A -85,B 0,C 180,E1 -12885.466,E2 -12885.466} C_VEL
LIN {X 0,Y 368.979,Z 242.526,A -85,B 0,C 180,E1 -12888.894,E2 -12888.894} C_VEL
LIN {X 0,Y 368.96,Z 242.525,A -85,B 0,C 180,E1 -12892.394,E2 -12892.394} C_VEL
LIN {X 0,Y 368.987,Z 242.52,A -85,B 0,C 180,E1 -12895.982,E2 -12895.982} C_VEL
LIN {X 0,Y 368.947,Z 242.53,A -85,B 0,C 180,E1 -12898.813,E2 -12898.813} C_VEL
LIN {X 0,Y 368.873,Z 242.535,A -85,B 0,C 180,E1 -12901.461,E2 -12901.461} C_VEL
LIN {X 0,Y 368.196,Z 242.622,A -85,B 0,C 180,E1 -12902.373,E2 -12902.373} C_VEL
LIN {X 0,Y 365.346,Z 242.974,A -85,B 0,C 180,E1 -12903.855,E2 -12903.855} C_VEL
LIN {X 0,Y 362.941,Z 243.276,A -85,B 0,C 180,E1 -12905.054,E2 -12905.054} C_VEL
LIN {X 0,Y 361.913,Z 243.402,A -85,B 0,C 180,E1 -12905.981,E2 -12905.981} C_VEL
LIN {X 0,Y 361.832,Z 243.409,A -85,B 0,C 180,E1 -12906.295,E2 -12906.295} C_VEL
LIN {X 0,Y 361.871,Z 243.407,A -85,B 0,C 180,E1 -12909.86,E2 -12909.86} C_VEL
LIN {X 0,Y 361.879,Z 243.409,A -85,B 0,C 180,E1 -12912.823,E2 -12912.823} C_VEL
LIN {X 0,Y 361.921,Z 243.401,A -85,B 0,C 180,E1 -12915.93,E2 -12915.93} C_VEL
LIN {X 0,Y 361.897,Z 243.403,A -85,B 0,C 180,E1 -12919.234,E2 -12919.234} C_VEL
LIN {X 0,Y 361.867,Z 243.408,A -85,B 0,C 180,E1 -12922.985,E2 -12922.985} C_VEL
LIN {X 0,Y 361.858,Z 243.411,A -85,B 0,C 180,E1 -12926.632,E2 -12926.632} C_VEL
LIN {X 0,Y 361.872,Z 243.407,A -85,B 0,C 180,E1 -12929.674,E2 -12929.674} C_VEL
LIN {X 0,Y 361.951,Z 243.397,A -85,B 0,C 180,E1 -12933.477,E2 -12933.477} C_VEL
LIN {X 0,Y 361.887,Z 243.404,A -85,B 0,C 180,E1 -12937.147,E2 -12937.147} C_VEL
LIN {X 0,Y 361.919,Z 243.401,A -85,B 0,C 180,E1 -12940.726,E2 -12940.726} C_VEL
LIN {X 0,Y 361.945,Z 243.401,A -85,B 0,C 180,E1 -12944.228,E2 -12944.228} C_VEL
LIN {X 0,Y 361.998,Z 243.392,A -85,B 0,C 180,E1 -12946.53,E2 -12946.53} C_VEL
LIN {X 0,Y 362.029,Z 243.392,A -85,B 0,C 180,E1 -12949.94,E2 -12949.94} C_VEL
LIN {X 0,Y 362.151,Z 243.373,A -85,B 0,C 180,E1 -12953.315,E2 -12953.315} C_VEL
LIN {X 0,Y 362.282,Z 243.36,A -85,B 0,C 180,E1 -12957.778,E2 -12957.778} C_VEL
LIN {X 0,Y 362.429,Z 243.34,A -85,B 0,C 180,E1 -12960.002,E2 -12960.002} C_VEL
LIN {X 0,Y 362.283,Z 243.357,A -85,B 0,C 180,E1 -12962.225,E2 -12962.225} C_VEL
LIN {X 0,Y 362.138,Z 243.373,A -85,B 0,C 180,E1 -12966.689,E2 -12966.689} C_VEL
LIN {X 0,Y 362.004,Z 243.392,A -85,B 0,C 180,E1 -12970.065,E2 -12970.065} C_VEL
LIN {X 0,Y 362.003,Z 243.393,A -85,B 0,C 180,E1 -12973.9,E2 -12973.9} C_VEL
LIN {X 0,Y 361.973,Z 243.395,A -85,B 0,C 180,E1 -12977.94,E2 -12977.94} C_VEL
LIN {X 0,Y 361.896,Z 243.407,A -85,B 0,C 180,E1 -12981.654,E2 -12981.654} C_VEL
LIN {X 0,Y 361.934,Z 243.404,A -85,B 0,C 180,E1 -12985.291,E2 -12985.291} C_VEL
LIN {X 0,Y 361.915,Z 243.403,A -85,B 0,C 180,E1 -12987.78,E2 -12987.78} C_VEL
LIN {X 0,Y 361.844,Z 243.412,A -85,B 0,C 180,E1 -12991.63,E2 -12991.63} C_VEL
LIN {X 0,Y 361.881,Z 243.41,A -85,B 0,C 180,E1 -12995.346,E2 -12995.346} C_VEL
LIN {X 0,Y 361.875,Z 243.411,A -85,B 0,C 180,E1 -12999.027,E2 -12999.027} C_VEL
LIN {X 0,Y 361.843,Z 243.41,A -85,B 0,C 180,E1 -13002.83,E2 -13002.83} C_VEL
LIN {X 0,Y 361.894,Z 243.59,A -85,B 0,C 180,E1 -13003.966,E2 -13003.966} C_VEL
LIN {X 0,Y 362.906,Z 249.019,A -85,B 0,C 180,E1 -13007.385,E2 -13007.385} C_VEL
LIN {X 0,Y 363.887,Z 254.394,A -85,B 0,C 180,E1 -13010.585,E2 -13010.585} C_VEL
LIN {X 0,Y 364.499,Z 259.208,A -85,B 0,C 180,E1 -13013.293,E2 -13013.293} C_VEL
LIN {X 0,Y 364.028,Z 264.621,A -85,B 0,C 180,E1 -13016.118,E2 -13016.118} C_VEL
LIN {X 0,Y 363.334,Z 270.684,A -85,B 0,C 180,E1 -13019.163,E2 -13019.163} C_VEL
LIN {X 0,Y 362.73,Z 277.066,A -85,B 0,C 180,E1 -13022.289,E2 -13022.289} C_VEL
LIN {X 0,Y 362.03,Z 284.737,A -85,B 0,C 180,E1 -13025.941,E2 -13025.941} C_VEL
LIN {X 0,Y 361.487,Z 292.429,A -85,B 0,C 180,E1 -13029.515,E2 -13029.515} C_VEL
LIN {X 0,Y 361.421,Z 293.599,A -85,B 0,C 180,E1 -13030.054,E2 -13030.054} C_VEL
LIN {X 0,Y 363.711,Z 307.302,A -85,B 0,C 180,E1 -13030.658,E2 -13030.658} C_VEL
LIN {X 0,Y 365.392,Z 319.932,A -85,B 0,C 180,E1 -13031.423,E2 -13031.423} C_VEL
LIN {X 0,Y 366.471,Z 331.104,A -85,B 0,C 180,E1 -13032.275,E2 -13032.275} C_VEL
LIN {X 0,Y 365.261,Z 343.461,A -85,B 0,C 180,E1 -13033.368,E2 -13033.368} C_VEL
LIN {X 0,Y 364.267,Z 353.674,A -85,B 0,C 180,E1 -13034.523,E2 -13034.523} C_VEL
LIN {X 0,Y 363.48,Z 362.384,A -85,B 0,C 180,E1 -13035.727,E2 -13035.727} C_VEL
LIN {X 0,Y 362.598,Z 370.729,A -85,B 0,C 180,E1 -13037.12,E2 -13037.12} C_VEL
LIN {X 0,Y 361.679,Z 378.902,A -85,B 0,C 180,E1 -13038.795,E2 -13038.795} C_VEL
LIN {X 0,Y 361.117,Z 385.492,A -85,B 0,C 180,E1 -13040.477,E2 -13040.477} C_VEL
LIN {X 0,Y 360.723,Z 390.733,A -85,B 0,C 180,E1 -13042.161,E2 -13042.161} C_VEL
LIN {X 0,Y 360.522,Z 394.767,A -85,B 0,C 180,E1 -13043.83,E2 -13043.83} C_VEL
LIN {X 0,Y 360.45,Z 397.797,A -85,B 0,C 180,E1 -13045.526,E2 -13045.526} C_VEL
LIN {X 0,Y 360.356,Z 399.241,A -85,B 0,C 180,E1 -13046.645,E2 -13046.645} C_VEL
LIN {X 0,Y 360.413,Z 400.261,A -85,B 0,C 180,E1 -13047.764,E2 -13047.764} C_VEL
LIN {X 0,Y 360.478,Z 400.885,A -85,B 0,C 180,E1 -13048.882,E2 -13048.882} C_VEL
LIN {X 0,Y 360.468,Z 401.11,A -85,B 0,C 180,E1 -13049.999,E2 -13049.999} C_VEL
LIN {X 0,Y 360.478,Z 400.907,A -85,B 0,C 180,E1 -13051.117,E2 -13051.117} C_VEL
LIN {X 0,Y 360.415,Z 400.281,A -85,B 0,C 180,E1 -13052.234,E2 -13052.234} C_VEL
LIN {X 0,Y 360.449,Z 397.846,A -85,B 0,C 180,E1 -13054.472,E2 -13054.472} C_VEL
LIN {X 0,Y 360.525,Z 394.83,A -85,B 0,C 180,E1 -13056.173,E2 -13056.173} C_VEL
LIN {X 0,Y 360.722,Z 390.85,A -85,B 0,C 180,E1 -13057.838,E2 -13057.838} C_VEL
LIN {X 0,Y 361.225,Z 384.712,A -85,B 0,C 180,E1 -13059.801,E2 -13059.801} C_VEL
LIN {X 0,Y 361.839,Z 378.004,A -85,B 0,C 180,E1 -13061.483,E2 -13061.483} C_VEL
LIN {X 0,Y 362.778,Z 369.711,A -85,B 0,C 180,E1 -13063.157,E2 -13063.157} C_VEL
LIN {X 0,Y 363.784,Z 360.18,A -85,B 0,C 180,E1 -13064.709,E2 -13064.709} C_VEL
LIN {X 0,Y 364.759,Z 349.731,A -85,B 0,C 180,E1 -13066.079,E2 -13066.079} C_VEL
LIN {X 0,Y 366.073,Z 337.874,A -85,B 0,C 180,E1 -13067.311,E2 -13067.311} C_VEL
LIN {X 0,Y 366.718,Z 330.114,A -85,B 0,C 180,E1 -13067.967,E2 -13067.967} C_VEL
LIN {X 0,Y 365.513,Z 317.711,A -85,B 0,C 180,E1 -13068.932,E2 -13068.932} C_VEL
LIN {X 0,Y 363.886,Z 305.096,A -85,B 0,C 180,E1 -13069.701,E2 -13069.701} C_VEL
LIN {X 0,Y 361.441,Z 292.204,A -85,B 0,C 180,E1 -13070.333,E2 -13070.333} C_VEL
LIN {X 0,Y 361.986,Z 284.037,A -85,B 0,C 180,E1 -13074.143,E2 -13074.143} C_VEL
LIN {X 0,Y 362.652,Z 276.628,A -85,B 0,C 180,E1 -13077.716,E2 -13077.716} C_VEL
LIN {X 0,Y 363.311,Z 270.407,A -85,B 0,C 180,E1 -13080.838,E2 -13080.838} C_VEL
LIN {X 0,Y 364.247,Z 263.066,A -85,B 0,C 180,E1 -13084.693,E2 -13084.693} C_VEL
LIN {X 0,Y 364.569,Z 259.535,A -85,B 0,C 180,E1 -13086.698,E2 -13086.698} C_VEL
LIN {X 0,Y 364.173,Z 256.114,A -85,B 0,C 180,E1 -13088.769,E2 -13088.769} C_VEL
LIN {X 0,Y 363.322,Z 251.46,A -85,B 0,C 180,E1 -13091.862,E2 -13091.862} C_VEL
LIN {X 0,Y 362.403,Z 246.233,A -85,B 0,C 180,E1 -13095.72,E2 -13095.72} C_VEL
LIN {X 0,Y 361.878,Z 243.41,A -85,B 0,C 180,E1 -13098.096,E2 -13098.096} C_VEL
LIN {X 0,Y 361.876,Z 243.409,A -85,B 0,C 180,E1 -13101.575,E2 -13101.575} C_VEL
LIN {X 0,Y 361.875,Z 243.41,A -85,B 0,C 180,E1 -13104.654,E2 -13104.654} C_VEL
LIN {X 0,Y 361.838,Z 243.414,A -85,B 0,C 180,E1 -13108.369,E2 -13108.369} C_VEL
LIN {X 0,Y 361.9,Z 243.404,A -85,B 0,C 180,E1 -13110.954,E2 -13110.954} C_VEL
LIN {X 0,Y 361.954,Z 243.4,A -85,B 0,C 180,E1 -13113.473,E2 -13113.473} C_VEL
LIN {X 0,Y 361.889,Z 243.405,A -85,B 0,C 180,E1 -13117.143,E2 -13117.143} C_VEL
LIN {X 0,Y 361.919,Z 243.404,A -85,B 0,C 180,E1 -13120.722,E2 -13120.722} C_VEL
LIN {X 0,Y 361.944,Z 243.398,A -85,B 0,C 180,E1 -13124.224,E2 -13124.224} C_VEL
LIN {X 0,Y 361.997,Z 243.393,A -85,B 0,C 180,E1 -13126.526,E2 -13126.526} C_VEL
LIN {X 0,Y 362.029,Z 243.39,A -85,B 0,C 180,E1 -13129.936,E2 -13129.936} C_VEL
LIN {X 0,Y 362.148,Z 243.376,A -85,B 0,C 180,E1 -13132.191,E2 -13132.191} C_VEL
LIN {X 0,Y 362.116,Z 243.381,A -85,B 0,C 180,E1 -13134.429,E2 -13134.429} C_VEL
LIN {X 0,Y 362.279,Z 243.357,A -85,B 0,C 180,E1 -13137.775,E2 -13137.775} C_VEL
LIN {X 0,Y 362.425,Z 243.341,A -85,B 0,C 180,E1 -13139.998,E2 -13139.998} C_VEL
LIN {X 0,Y 362.278,Z 243.361,A -85,B 0,C 180,E1 -13142.222,E2 -13142.222} C_VEL
LIN {X 0,Y 362.167,Z 243.374,A -85,B 0,C 180,E1 -13146.684,E2 -13146.684} C_VEL
LIN {X 0,Y 362.063,Z 243.388,A -85,B 0,C 180,E1 -13148.931,E2 -13148.931} C_VEL
LIN {X 0,Y 361.887,Z 243.415,A -85,B 0,C 180,E1 -13151.196,E2 -13151.196} C_VEL
LIN {X 0,Y 361.834,Z 245.231,A -85,B 0,C 180,E1 -13153.797,E2 -13153.797} C_VEL
LIN {X 0,Y 361.625,Z 248.464,A -85,B 0,C 180,E1 -13157.773,E2 -13157.773} C_VEL
LIN {X 0,Y 361.387,Z 251.765,A -85,B 0,C 180,E1 -13161.682,E2 -13161.682} C_VEL
LIN {X 0,Y 361.244,Z 254.941,A -85,B 0,C 180,E1 -13165.339,E2 -13165.339} C_VEL
LIN {X 0,Y 361.197,Z 256.361,A -85,B 0,C 180,E1 -13166.758,E2 -13166.758} C_VEL
LIN {X 0,Y 365.37,Z 269.748,A -85,B 0,C 180,E1 -13167.607,E2 -13167.607} C_VEL
LIN {X 0,Y 368.174,Z 281.466,A -85,B 0,C 180,E1 -13168.501,E2 -13168.501} C_VEL
LIN {X 0,Y 368.406,Z 284.422,A -85,B 0,C 180,E1 -13168.734,E2 -13168.734} C_VEL
LIN {X 0,Y 367.472,Z 295.727,A -85,B 0,C 180,E1 -13169.643,E2 -13169.643} C_VEL
LIN {X 0,Y 366.35,Z 307.428,A -85,B 0,C 180,E1 -13170.847,E2 -13170.847} C_VEL
LIN {X 0,Y 365.274,Z 317.531,A -85,B 0,C 180,E1 -13172.161,E2 -13172.161} C_VEL
LIN {X 0,Y 364.238,Z 326.62,A -85,B 0,C 180,E1 -13173.618,E2 -13173.618} C_VEL
LIN {X 0,Y 363.356,Z 334.253,A -85,B 0,C 180,E1 -13175.126,E2 -13175.126} C_VEL
LIN {X 0,Y 362.386,Z 341.626,A -85,B 0,C 180,E1 -13176.953,E2 -13176.953} C_VEL
LIN {X 0,Y 361.599,Z 347.928,A -85,B 0,C 180,E1 -13178.975,E2 -13178.975} C_VEL
LIN {X 0,Y 361.197,Z 351.811,A -85,B 0,C 180,E1 -13180.639,E2 -13180.639} C_VEL
LIN {X 0,Y 360.877,Z 354.612,A -85,B 0,C 180,E1 -13182.266,E2 -13182.266} C_VEL
LIN {X 0,Y 360.53,Z 357.035,A -85,B 0,C 180,E1 -13184.566,E2 -13184.566} C_VEL
LIN {X 0,Y 360.371,Z 357.729,A -85,B 0,C 180,E1 -13186.181,E2 -13186.181} C_VEL
LIN {X 0,Y 360.372,Z 357.272,A -85,B 0,C 180,E1 -13188.467,E2 -13188.467} C_VEL
LIN {X 0,Y 360.493,Z 356.05,A -85,B 0,C 180,E1 -13189.959,E2 -13189.959} C_VEL
LIN {X 0,Y 360.704,Z 354.151,A -85,B 0,C 180,E1 -13191.429,E2 -13191.429} C_VEL
LIN {X 0,Y 360.97,Z 351.379,A -85,B 0,C 180,E1 -13192.96,E2 -13192.96} C_VEL
LIN {X 0,Y 361.403,Z 346.986,A -85,B 0,C 180,E1 -13194.756,E2 -13194.756} C_VEL
LIN {X 0,Y 361.937,Z 341.039,A -85,B 0,C 180,E1 -13196.607,E2 -13196.607} C_VEL
LIN {X 0,Y 362.756,Z 333.364,A -85,B 0,C 180,E1 -13198.474,E2 -13198.474} C_VEL
LIN {X 0,Y 363.621,Z 324.664,A -85,B 0,C 180,E1 -13200.141,E2 -13200.141} C_VEL
LIN {X 0,Y 364.562,Z 315.017,A -85,B 0,C 180,E1 -13201.631,E2 -13201.631} C_VEL
LIN {X 0,Y 365.484,Z 305.481,A -85,B 0,C 180,E1 -13202.827,E2 -13202.827} C_VEL
LIN {X 0,Y 366.406,Z 294.333,A -85,B 0,C 180,E1 -13203.952,E2 -13203.952} C_VEL
LIN {X 0,Y 367.292,Z 282.627,A -85,B 0,C 180,E1 -13204.878,E2 -13204.878} C_VEL
LIN {X 0,Y 367.144,Z 279.69,A -85,B 0,C 180,E1 -13205.095,E2 -13205.095} C_VEL
LIN {X 0,Y 364.394,Z 267.288,A -85,B 0,C 180,E1 -13205.957,E2 -13205.957} C_VEL
LIN {X 0,Y 360.881,Z 253.956,A -85,B 0,C 180,E1 -13206.697,E2 -13206.697} C_VEL
LIN {X 0,Y 360.972,Z 250.053,A -85,B 0,C 180,E1 -13210.672,E2 -13210.672} C_VEL
LIN {X 0,Y 361.088,Z 246.679,A -85,B 0,C 180,E1 -13214.188,E2 -13214.188} C_VEL
LIN {X 0,Y 361.291,Z 243.484,A -85,B 0,C 180,E1 -13217.645,E2 -13217.645} C_VEL
LIN {X 0,Y 361.784,Z 243.42,A -85,B 0,C 180,E1 -13221.06,E2 -13221.06} C_VEL
LIN {X 0,Y 362.101,Z 243.383,A -85,B 0,C 180,E1 -13223.313,E2 -13223.313} C_VEL
LIN {X 0,Y 362.268,Z 243.359,A -85,B 0,C 180,E1 -13227.777,E2 -13227.777} C_VEL
LIN {X 0,Y 362.414,Z 243.339,A -85,B 0,C 180,E1 -13230.001,E2 -13230.001} C_VEL
LIN {X 0,Y 362.268,Z 243.357,A -85,B 0,C 180,E1 -13232.224,E2 -13232.224} C_VEL
LIN {X 0,Y 362.157,Z 243.372,A -85,B 0,C 180,E1 -13236.687,E2 -13236.687} C_VEL
LIN {X 0,Y 362.06,Z 243.387,A -85,B 0,C 180,E1 -13238.934,E2 -13238.934} C_VEL
LIN {X 0,Y 361.951,Z 243.397,A -85,B 0,C 180,E1 -13242.333,E2 -13242.333} C_VEL
LIN {X 0,Y 361.947,Z 243.399,A -85,B 0,C 180,E1 -13244.622,E2 -13244.622} C_VEL
LIN {X 0,Y 361.947,Z 243.397,A -85,B 0,C 180,E1 -13248.1,E2 -13248.1} C_VEL
LIN {X 0,Y 361.912,Z 243.402,A -85,B 0,C 180,E1 -13251.652,E2 -13251.652} C_VEL
LIN {X 0,Y 361.917,Z 243.403,A -85,B 0,C 180,E1 -13255.291,E2 -13255.291} C_VEL
LIN {X 0,Y 361.901,Z 243.403,A -85,B 0,C 180,E1 -13257.78,E2 -13257.78} C_VEL
LIN {X 0,Y 361.828,Z 243.412,A -85,B 0,C 180,E1 -13261.457,E2 -13261.457} C_VEL
LIN {X 0,Y 361.843,Z 243.412,A -85,B 0,C 180,E1 -13264.282,E2 -13264.282} C_VEL
LIN {X 0,Y 361.832,Z 243.409,A -85,B 0,C 180,E1 -13266.295,E2 -13266.295} C_VEL
LIN {X 0,Y 361.181,Z 243.495,A -85,B 0,C 180,E1 -13267.224,E2 -13267.224} C_VEL
LIN {X 0,Y 358.372,Z 243.847,A -85,B 0,C 180,E1 -13268.737,E2 -13268.737} C_VEL
LIN {X 0,Y 355.973,Z 244.146,A -85,B 0,C 180,E1 -13269.96,E2 -13269.96} C_VEL
LIN {X 0,Y 354.923,Z 244.275,A -85,B 0,C 180,E1 -13270.906,E2 -13270.906} C_VEL
LIN {X 0,Y 354.826,Z 244.284,A -85,B 0,C 180,E1 -13271.226,E2 -13271.226} C_VEL
LIN {X 0,Y 354.879,Z 244.283,A -85,B 0,C 180,E1 -13274.529,E2 -13274.529} C_VEL
LIN {X 0,Y 354.832,Z 244.283,A -85,B 0,C 180,E1 -13277.672,E2 -13277.672} C_VEL
LIN {X 0,Y 354.83,Z 244.287,A -85,B 0,C 180,E1 -13280.671,E2 -13280.671} C_VEL
LIN {X 0,Y 354.816,Z 244.29,A -85,B 0,C 180,E1 -13284.303,E2 -13284.303} C_VEL
LIN {X 0,Y 354.793,Z 244.288,A -85,B 0,C 180,E1 -13287.67,E2 -13287.67} C_VEL
LIN {X 0,Y 354.864,Z 244.282,A -85,B 0,C 180,E1 -13290.623,E2 -13290.623} C_VEL
LIN {X 0,Y 354.896,Z 244.28,A -85,B 0,C 180,E1 -13294.175,E2 -13294.175} C_VEL
LIN {X 0,Y 354.832,Z 244.287,A -85,B 0,C 180,E1 -13297.896,E2 -13297.896} C_VEL
LIN {X 0,Y 354.922,Z 244.276,A -85,B 0,C 180,E1 -13301.894,E2 -13301.894} C_VEL
LIN {X 0,Y 354.942,Z 244.275,A -85,B 0,C 180,E1 -13305.983,E2 -13305.983} C_VEL
LIN {X 0,Y 354.976,Z 244.269,A -85,B 0,C 180,E1 -13309.738,E2 -13309.738} C_VEL
LIN {X 0,Y 355.114,Z 244.249,A -85,B 0,C 180,E1 -13313.182,E2 -13313.182} C_VEL
LIN {X 0,Y 355.246,Z 244.237,A -85,B 0,C 180,E1 -13317.734,E2 -13317.734} C_VEL
LIN {X 0,Y 355.399,Z 244.216,A -85,B 0,C 180,E1 -13320.002,E2 -13320.002} C_VEL
LIN {X 0,Y 355.246,Z 244.233,A -85,B 0,C 180,E1 -13322.269,E2 -13322.269} C_VEL
LIN {X 0,Y 355.102,Z 244.249,A -85,B 0,C 180,E1 -13326.822,E2 -13326.822} C_VEL
LIN {X 0,Y 354.96,Z 244.268,A -85,B 0,C 180,E1 -13330.266,E2 -13330.266} C_VEL
LIN {X 0,Y 354.948,Z 244.27,A -85,B 0,C 180,E1 -13334.02,E2 -13334.02} C_VEL
LIN {X 0,Y 354.928,Z 244.272,A -85,B 0,C 180,E1 -13338.11,E2 -13338.11} C_VEL
LIN {X 0,Y 354.839,Z 244.283,A -85,B 0,C 180,E1 -13342.107,E2 -13342.107} C_VEL
LIN {X 0,Y 354.905,Z 244.276,A -85,B 0,C 180,E1 -13345.829,E2 -13345.829} C_VEL
LIN {X 0,Y 354.825,Z 244.286,A -85,B 0,C 180,E1 -13349.683,E2 -13349.683} C_VEL
LIN {X 0,Y 354.813,Z 244.287,A -85,B 0,C 180,E1 -13353.703,E2 -13353.703} C_VEL
LIN {X 0,Y 354.804,Z 244.287,A -85,B 0,C 180,E1 -13356.46,E2 -13356.46} C_VEL
LIN {X 0,Y 354.832,Z 244.286,A -85,B 0,C 180,E1 -13359.424,E2 -13359.424} C_VEL
LIN {X 0,Y 354.824,Z 244.294,A -85,B 0,C 180,E1 -13363.468,E2 -13363.468} C_VEL
LIN {X 0,Y 355.799,Z 249.682,A -85,B 0,C 180,E1 -13366.96,E2 -13366.96} C_VEL
LIN {X 0,Y 356.795,Z 254.975,A -85,B 0,C 180,E1 -13370.195,E2 -13370.195} C_VEL
LIN {X 0,Y 357.49,Z 260.111,A -85,B 0,C 180,E1 -13373.143,E2 -13373.143} C_VEL
LIN {X 0,Y 357.093,Z 264.992,A -85,B 0,C 180,E1 -13375.754,E2 -13375.754} C_VEL
LIN {X 0,Y 356.3,Z 271.59,A -85,B 0,C 180,E1 -13379.146,E2 -13379.146} C_VEL
LIN {X 0,Y 355.562,Z 278.942,A -85,B 0,C 180,E1 -13382.808,E2 -13382.808} C_VEL
LIN {X 0,Y 354.938,Z 285.756,A -85,B 0,C 180,E1 -13386.129,E2 -13386.129} C_VEL
LIN {X 0,Y 354.403,Z 293.263,A -85,B 0,C 180,E1 -13389.674,E2 -13389.674} C_VEL
LIN {X 0,Y 356.64,Z 306.661,A -85,B 0,C 180,E1 -13390.279,E2 -13390.279} C_VEL
LIN {X 0,Y 358.3,Z 319.041,A -85,B 0,C 180,E1 -13391.041,E2 -13391.041} C_VEL
LIN {X 0,Y 359.564,Z 330.329,A -85,B 0,C 180,E1 -13391.923,E2 -13391.923} C_VEL
LIN {X 0,Y 358.562,Z 341.342,A -85,B 0,C 180,E1 -13392.901,E2 -13392.901} C_VEL
LIN {X 0,Y 357.536,Z 351.491,A -85,B 0,C 180,E1 -13394.026,E2 -13394.026} C_VEL
LIN {X 0,Y 356.548,Z 361.784,A -85,B 0,C 180,E1 -13395.444,E2 -13395.444} C_VEL
LIN {X 0,Y 355.649,Z 370.16,A -85,B 0,C 180,E1 -13396.864,E2 -13396.864} C_VEL
LIN {X 0,Y 354.672,Z 378.357,A -85,B 0,C 180,E1 -13398.57,E2 -13398.57} C_VEL
LIN {X 0,Y 354.087,Z 384.97,A -85,B 0,C 180,E1 -13400.287,E2 -13400.287} C_VEL
LIN {X 0,Y 353.658,Z 390.233,A -85,B 0,C 180,E1 -13402.003,E2 -13402.003} C_VEL
LIN {X 0,Y 353.44,Z 394.583,A -85,B 0,C 180,E1 -13403.85,E2 -13403.85} C_VEL
